(* IEC 61131-3 sources: volt/packages/volt-lsp-iec/test-corpus/pro2193/Device/Plc Logic/Application/09 Misc/Library Manager/L_MC1P_MotionControlBasic (part 7) *)

(* ---- L_MC1P_RESETMASTER_ETC.pou ---- *)
FUNCTION_BLOCK L_MC1P_RESETMASTER_ETC
VAR_INPUT
	XEXECUTE : BOOL;
	PSLAVE : POINTER TO ETCSlave;
END_VAR
VAR_OUTPUT
	XDONE : BOOL;
	XERROR : BOOL;
	XBUSY : BOOL;
	DWERROR : DWORD;
END_VAR
VAR
	XEXECUTEOLD : BOOL;
	WACTMASTERSTATE : INT;
	SETMASTERSTATE : L_ETC.L_ETC_SetMasterState;
	PMASTER : POINTER TO L_ETC.L_IODrvEtherCAT;
END_VAR
END_FUNCTION_BLOCK

METHOD ACYCLICACTION
END_METHOD

(* ---- L_MC1P_SAFETYCONTROLDECODER.pou ---- *)
FUNCTION_BLOCK L_MC1P_SAFETYCONTROLDECODER
VAR_INPUT
	XENABLE : BOOL;
	DWCONTROL : DWORD;
END_VAR
VAR_OUTPUT
	XBUSY : BOOL;
	XERROR : BOOL;
	EERRORID : L_IE1P_Error;
	XSTO_ACTIVE : BOOL;
	XSS1_ACTIVE : BOOL;
	XSS2_ACTIVE : BOOL;
	XSOS_ACTIVE : BOOL;
	XSLS1_ACTIVE : BOOL;
	XSLS2_ACTIVE : BOOL;
	XSLS3_ACTIVE : BOOL;
	XSLS4_ACTIVE : BOOL;
	XSDIPOS_ACTIVE : BOOL;
	XSDINEG_ACTIVE : BOOL;
	XSLI_ACTIVE : BOOL;
	XSSE_ACTIVE : BOOL;
	XES_ACTIVE : BOOL;
	XOMS_ACTIVE : BOOL;
	XRMS_ACTIVE : BOOL;
	XSBC_ACTIVE : BOOL;
	XMUT_ACTIVE : BOOL;
END_VAR
END_FUNCTION_BLOCK

(* ---- L_MC1P_SAFETYCONTROLENCODER.pou ---- *)
FUNCTION_BLOCK L_MC1P_SAFETYCONTROLENCODER
VAR_INPUT
	XENABLE : BOOL;
	XSTO_ACTIVE : BOOL;
	XSS1_ACTIVE : BOOL;
	XSS2_ACTIVE : BOOL;
	XSOS_ACTIVE : BOOL;
	XSLS1_ACTIVE : BOOL;
	XSLS2_ACTIVE : BOOL;
	XSLS3_ACTIVE : BOOL;
	XSLS4_ACTIVE : BOOL;
	XSDIPOS_ACTIVE : BOOL;
	XSDINEG_ACTIVE : BOOL;
	XSLI_ACTIVE : BOOL;
	XSSE_ACTIVE : BOOL;
	XES_ACTIVE : BOOL;
	XOMS_ACTIVE : BOOL;
	XRMS_ACTIVE : BOOL;
	XSBC_ACTIVE : BOOL;
	XMUT_ACTIVE : BOOL;
END_VAR
VAR_OUTPUT
	XBUSY : BOOL;
	XERROR : BOOL;
	EERRORID : L_IE1P_Error;
	DWCONTROL : DWORD;
END_VAR
END_FUNCTION_BLOCK

(* ---- L_MC1P_SAFETYIOSTATEDECODER.pou ---- *)
FUNCTION_BLOCK L_MC1P_SAFETYIOSTATEDECODER
VAR_INPUT
	XENABLE : BOOL;
	DWIOSTATE : DWORD;
END_VAR
VAR_OUTPUT
	XBUSY : BOOL;
	XERROR : BOOL;
	EERRORID : L_IE1P_Error;
	XSDIN1 : BOOL;
	XSDIN2 : BOOL;
	XSDIN3 : BOOL;
	XSDIN4 : BOOL;
	XAIS_DIGIN : BOOL;
	XAIE_DIGIN : BOOL;
	XIRS_DIGIN : BOOL;
	XIRL_DIGIN : BOOL;
	XAIS_SBUS : BOOL;
	XAIE_SBUS : BOOL;
	XSHOMSTART_SBUS : BOOL;
	XSHOMLOAD_SBUS : BOOL;
	XSDOUT1 : BOOL;
	XSDIN1A : BOOL;
	XSDIN1B : BOOL;
	XSDIN2A : BOOL;
	XSDIN2B : BOOL;
	XSDIN3A : BOOL;
	XSDIN3B : BOOL;
	XSDIN4A : BOOL;
	XSDIN4B : BOOL;
	XSDOUT1A : BOOL;
	XSDOUT1B : BOOL;
END_VAR
END_FUNCTION_BLOCK

(* ---- L_MC1P_SAFETYREADSTATUSWORDS.pou ---- *)
FUNCTION_BLOCK L_MC1P_SAFETYREADSTATUSWORDS EXTENDS L_MC1P_Template
VAR_INPUT
	XENABLE : BOOL;
END_VAR
VAR_OUTPUT
	XVALID : BOOL;
	XBUSY : BOOL;
	XERROR : BOOL;
	EERRORID : L_IE1P_Error;
	DWCONTROL : DWORD;
	DWSTATE : DWORD;
	DWIOSTATE : DWORD;
END_VAR
VAR
	XENABLEOLD : BOOL;
END_VAR
END_FUNCTION_BLOCK

(* ---- L_MC1P_SAFETYSTATEDECODER.pou ---- *)
FUNCTION_BLOCK L_MC1P_SAFETYSTATEDECODER
VAR_INPUT
	XENABLE : BOOL;
	DWSTATE : DWORD;
END_VAR
VAR_OUTPUT
	XBUSY : BOOL;
	XERROR : BOOL;
	EERRORID : L_IE1P_Error;
	XSLS1_OBSERVED : BOOL;
	XSLS2_OBSERVED : BOOL;
	XSLS3_OBSERVED : BOOL;
	XSLS4_OBSERVED : BOOL;
	XSMS_OBSERVED : BOOL;
	XSSM_WITHINLIMITS : BOOL;
	XSDIPOS_OBSERVED : BOOL;
	XSDINEG_OBSERVED : BOOL;
	XSLP1_OBSERVED : BOOL;
	XSLP2_OBSERVED : BOOL;
	XSLP3_OBSERVED : BOOL;
	XSLP4_OBSERVED : BOOL;
	XSCA1_WITHINLIMITS : BOOL;
	XSCA2_WITHINLIMITS : BOOL;
	XSCA3_WITHINLIMITS : BOOL;
	XSCA4_WITHINLIMITS : BOOL;
	XPDSSPOS_OBSERVED : BOOL;
	XPDSSNEG_OBSERVED : BOOL;
	XSOS_OBSERVED : BOOL;
	XSBC_ACTIVATED : BOOL;
	XSHOM_ACTIVE : BOOL;
	XSHOM_AVAILABLE : BOOL;
	XSAFESPEED_OK : BOOL;
	XSPEEDEQ0 : BOOL;
	XPOSDIRECTION : BOOL;
	XSLIPGT25 : BOOL;
	XSLIPGT50 : BOOL;
	XSLIPGT75 : BOOL;
	XERRORACTIVE : BOOL;
END_VAR
END_FUNCTION_BLOCK

(* ---- L_MC1P_SETAXISREFMASTERVALUES.pou ---- *)
FUNCTION_BLOCK L_MC1P_SETAXISREFMASTERVALUES
VAR_INPUT
	LRSETPOSIN : LREAL;
	LRSETVELIN : LREAL;
	LRSETACCIN : LREAL;
	LRTORQUEIN : LREAL;
	LRCYCLELENGTH : LREAL;
	ETRAVERSINGRANGE : L_MC1P_TraversingRange;
	XINTERPOLATEINPUTS : BOOL;
	LRINPUTCYCLETIME : LREAL := 0.001;
	EINTERPOLATIONMODE : L_MC1P_InterpolationMode := L_MC1P_InterpolationMode.linear;
	WDIRECTION : WORD;
	XACTIVATETELEGRAMLOSSDETECTION : BOOL;
	XSYNCPROCESSDATAEXPECTED : BOOL;
	XSYNCPROCESSDATAVALID : BOOL;
END_VAR
VAR_OUTPUT
	MASTERVALUES : L_MC1P_IAXIS_REF_MASTERVALUES;
	LRSETPOSOUT : LREAL;
	LRSETVELOUT : LREAL;
	LRSETACCOUT : LREAL;
	LRTORQUEOUT : LREAL;
END_VAR
VAR
	XINITDONE : BOOL := FALSE;
	LRSETPOSINOLD : LREAL;
	LRSETVELINOLD : LREAL;
	LRSETACCINOLD : LREAL;
	LRTORQUEINOLD : LREAL;
	LRSETPOSSTART : LREAL;
	LRSETVELSTART : LREAL;
	LRSETACCSTART : LREAL;
	LRTORQUESTART : LREAL;
	LRSETPOSEND : LREAL;
	LRSETVELEND : LREAL;
	LRSETACCEND : LREAL;
	LRTORQUEEND : LREAL;
	LRTASKCYCLE : LREAL := 0.001;
	LRINVTASKCYCLE : LREAL := 1000;
	LRACTCYCLE : LREAL;
	LRMAXCYCLE : LREAL;
	LRINVMAXCYCLE : LREAL;
	XSTARTINTERPOLATION : BOOL;
	LRPOSDIFF : LREAL;
	LRPOSDIFFOLD : LREAL;
	LRSETPOSSTARTOLD : LREAL;
	LRACC : LREAL;
	LRVEL : LREAL;
	FB_GETDIRECTION : L_MC1P_GetDirection;
	WEXTRAPOLATIONCOUNTER : WORD;
	WINTERPOLATIONCOUNTER : WORD;
	POSV : LREAL;
	C_COUNTERLIMIT : WORD := 1000;
	ACTACCELERATION : LREAL;
	ACTPOSITION : LREAL;
	ACTTORQUE : LREAL;
	ACTVELOCITY : LREAL;
	CYCLELENGTH : LREAL;
	FEEDCONSTANT : LREAL;
	GETMASTERID : POINTER TO BYTE;
	SETACCELERATIONFORSYNC : LREAL;
	SETPOSITIONFORSYNC : LREAL;
	SETTORQUEFORSYNC : LREAL;
	SETVELOCITYFORSYNC : LREAL;
	TASKCYCLE : LREAL;
	TRAVERSINGRANGE : L_MC1P_TraversingRange;
END_VAR
END_FUNCTION_BLOCK

METHOD GETDIRECTION : WORD
VAR_INPUT
	VALUESOURCE : MC_SOURCE;
END_VAR
END_METHOD

METHOD GETMASTERERROR : BOOL
VAR_OUTPUT
	EERRORID : L_IE1P_Error;
END_VAR
END_METHOD

METHOD GETSTEADYSTATE : POINTER TO L_MC1P_SteadyState
END_METHOD

METHOD FB_INIT : BOOL
VAR_INPUT
	BINITRETAINS : BOOL;
	BINCOPYCODE : BOOL;
END_VAR
END_METHOD

(* ---- L_MC1P_SETBASICPARAMETER.pou ---- *)
FUNCTION_BLOCK L_MC1P_SETBASICPARAMETER EXTENDS L_MC1P_Template
VAR_INPUT
	XENABLE : BOOL;
	XSETJOGPARAMETER : BOOL;
	LRJOGVEL : LREAL := 360;
	LRJOGACC : LREAL := 360;
	LRJOGDEC : LREAL := 1440;
	LRJOGJERK : LREAL := 0;
	XSETHALTPARAMETER : BOOL;
	LRHALTDEC : LREAL := 1800;
	LRHALTJERK : LREAL := 0;
	XSETQSPAPPLPARAMETER : BOOL;
	LRQSPAPPLDEC : LREAL := 3600.0;
	LRQSPAPPLJERK : LREAL := 0;
	XSETHOMEPOSITION : BOOL;
	LRHOMEPOSITION : LREAL;
	XSETHOMEPARAMETER : BOOL;
	SCHOMEPARAMETER : L_MC1P_HomeParameter := STRUCT(eHomeMode := L_MC1P_HomeMode.SetPositionDirect, eHomeStopMode := L_MC1P_HomeStopMode.StopPositioning, lrTargetPosition := 0, lrVelocity1 := 360.0, lrVelocity2 := 0, lrAcceleration1 := 720.0, lrAcceleration2 := 360.0, lrJerk := 7200.0, rTorqueLimit := 0.1, rTorqueTime := 1.0, dwTPConfig := 1, eStopModeDirection := MC_DIRECTION.mcCurrentDirection);
END_VAR
VAR_OUTPUT
	XBUSY : BOOL;
	XERROR : BOOL;
	EERRORID : L_IE1P_Error;
END_VAR
VAR
	ICACHEARRAYINITIDX : INT := -1;
	ICACHEARRAYFIRSTIDX : INT := 0;
	ICACHEARRAYLASTIDX : INT := 15;
	ADIRBPARAMETERS : ARRAY [iCacheArrayFirstIdx..iCacheArrayLastIdx] OF DINT;
	ALRRBVALUES : ARRAY [iCacheArrayFirstIdx..iCacheArrayLastIdx] OF LREAL;
	IRBACTIDX : INT := -1;
END_VAR
END_FUNCTION_BLOCK

METHOD SETBASICPARAMETER : DWORD
END_METHOD

METHOD WRITEPARAM : BOOL
VAR_INPUT
	PARAMETER : DINT;
	LRVALUE : LREAL;
	EWRITEERRORID : L_IE1P_Error;
END_VAR
END_METHOD

(* ---- L_MC1P_SETCONTROLMODE.pou ---- *)
FUNCTION_BLOCK L_MC1P_SETCONTROLMODE EXTENDS L_MC1P_Template
VAR_INPUT
	XEXECUTE : BOOL;
	ECONTROLMODE : L_MC1P_ControlModeSet := L_MC1P_ControlModeSet.PosCtrlDrive;
	XKEEPACTPOSPRIORFDB : BOOL := FALSE;
	XRESTARTPOSITIONING : BOOL := FALSE;
END_VAR
VAR_OUTPUT
	XDONE : BOOL;
	XBUSY : BOOL;
	XERROR : BOOL;
	EERRORID : L_IE1P_Error;
END_VAR
VAR
	FBSETCONTROLMODEINTERN : L_MC1P_SetControlMode_Internal;
END_VAR
END_FUNCTION_BLOCK

(* ---- L_MC1P_SETCONTROLMODE_INTERNAL.pou ---- *)
FUNCTION_BLOCK L_MC1P_SETCONTROLMODE_INTERNAL EXTENDS L_MC1P_Template_IntFB
VAR_INPUT
	XEXECUTE : BOOL;
	ECONTROLMODE : L_MC1P_ControlModeSet := L_MC1P_ControlModeSet.PosCtrlDrive;
	XKEEPACTPOSPRIORFDB : BOOL := FALSE;
	XRESTARTPOSITIONING : BOOL := FALSE;
END_VAR
VAR_OUTPUT
	XDONE : BOOL;
	XBUSY : BOOL;
	XERROR : BOOL;
	EERRORID : L_IE1P_Error;
END_VAR
VAR
	XEXECUTEOLD : BOOL;
	XRESETOUTPUT : BOOL;
END_VAR
END_FUNCTION_BLOCK

METHOD MAIN
VAR_IN_OUT
	AXIS : AXIS_REF;
	FBBASE : L_MC1P_Template_ForAxis;
END_VAR
END_METHOD

(* ---- L_MC1P_SETDCBRAKE.pou ---- *)
FUNCTION_BLOCK L_MC1P_SETDCBRAKE EXTENDS L_MC1P_Template
VAR_INPUT
	XENABLE : BOOL;
END_VAR
VAR_OUTPUT
	XBUSY : BOOL;
	XACTIVE : BOOL;
	XERROR : BOOL;
	EERRORID : L_IE1P_Error;
END_VAR
VAR
	XENABLEOLD : BOOL;
END_VAR
END_FUNCTION_BLOCK

(* ---- L_MC1P_SETEXTERNALENCODER.pou ---- *)
FUNCTION_BLOCK L_MC1P_SETEXTERNALENCODER EXTENDS L_MC1P_Template
VAR_INPUT
	ENCODER : L_MC1P_IEncoderInterface;
	XEXECUTE : BOOL;
END_VAR
VAR_OUTPUT
	XDONE : BOOL;
	XBUSY : BOOL;
	XERROR : BOOL;
	EERRORID : L_IE1P_Error;
END_VAR
VAR
	XEXECUTEOLD : BOOL;
	PAXISREALDRIVE : POINTER TO _AXIS_REF_REAL;
	PAXISREAL : POINTER TO _AXIS_REF_REAL;
	PXDUMMY : POINTER TO BOOL;
	PSDUMMY : POINTER TO STRING;
END_VAR
END_FUNCTION_BLOCK

(* ---- L_MC1P_SETFASTSTOP.pou ---- *)
FUNCTION_BLOCK L_MC1P_SETFASTSTOP EXTENDS L_MC1P_Template
VAR_INPUT
	XENABLE : BOOL;
END_VAR
VAR_OUTPUT
	XBUSY : BOOL;
	XACTIVE : BOOL;
	XERROR : BOOL;
	EERRORID : L_IE1P_Error;
END_VAR
VAR
	XENABLEOLD : BOOL;
	FBSETFASTSTOP : L_MC1P_SetFastStop_Internal;
END_VAR
END_FUNCTION_BLOCK

(* ---- L_MC1P_SETFASTSTOP_INTERNAL.pou ---- *)
FUNCTION_BLOCK L_MC1P_SETFASTSTOP_INTERNAL EXTENDS L_MC1P_Template_IntFB
VAR_INPUT
	XENABLE : BOOL;
END_VAR
VAR_OUTPUT
	XBUSY : BOOL;
	XACTIVE : BOOL;
	XERROR : BOOL;
	EERRORID : L_IE1P_Error;
END_VAR
VAR
	XENABLEOLD : BOOL;
END_VAR
END_FUNCTION_BLOCK

METHOD MAIN
VAR_IN_OUT
	AXIS : AXIS_REF;
	FBBASE : L_MC1P_Template_ForAxis;
END_VAR
END_METHOD

(* ---- L_MC1P_SETINERTIAADAPTVALUE.pou ---- *)
FUNCTION_BLOCK L_MC1P_SETINERTIAADAPTVALUE EXTENDS L_MC1P_Template
VAR_INPUT
	XENABLE : BOOL;
	LRINERTIAADAPTVALUE : LREAL := 1.0;
END_VAR
VAR_OUTPUT
	XBUSY : BOOL;
	XERROR : BOOL;
	EERRORID : L_IE1P_Error;
END_VAR
VAR
	PAXIS : POINTER TO _AXIS_REF_REAL;
	XENABLEOLD : BOOL;
END_VAR
END_FUNCTION_BLOCK

(* ---- L_MC1P_SETOVERRIDE_INTERNAL.pou ---- *)
FUNCTION_BLOCK L_MC1P_SETOVERRIDE_INTERNAL EXTENDS L_MC1P_Template_IntFB
VAR_INPUT
	ENABLE : BOOL;
	VELFACTOR : LREAL := 1.0;
	ACCFACTOR : LREAL := 1.0;
	JERKFACTOR : LREAL := 1.0;
END_VAR
VAR_OUTPUT
	ENABLED : BOOL;
	BUSY : BOOL;
	ERROR : BOOL;
	ERRORID : L_IE1P_Error;
END_VAR
VAR
	XENABLEOLD : BOOL;
	WDATAOLD : WORD;
END_VAR
END_FUNCTION_BLOCK

METHOD MAIN
VAR_IN_OUT
	AXIS : AXIS_REF;
	FBBASE : L_MC1P_Template_ForAxis;
END_VAR
END_METHOD

(* ---- L_MC1P_SETPOSCTRLADAPTVALUE.pou ---- *)
FUNCTION_BLOCK L_MC1P_SETPOSCTRLADAPTVALUE EXTENDS L_MC1P_Template
VAR_INPUT
	XENABLE : BOOL;
	LRPOSCTRLADAPTVALUE : LREAL := 1.0;
	EMODE : L_MC1P_PosCtrlAdaptMode := L_MC1P_PosCtrlAdaptMode.MotorAndLoad;
END_VAR
VAR_OUTPUT
	XBUSY : BOOL;
	XERROR : BOOL;
	EERRORID : L_IE1P_Error;
END_VAR
VAR
	ISTATE : INT := 0;
	DNPOSCTRLADAPTVAL : DINT;
	DNPOSCTRLADAPTVALOLD : DINT := 100;
	BYSDORETRYCOUNTER : BYTE;
	XWAITFORPARAMETERWRITEDONE : BOOL;
	WRITEPARAMETER : L_DCO_WriteDriveParameter;
	XCHECKCONFIG : BOOL;
	XUSEPDOINTERFACE : BOOL;
	WINDEX : WORD;
	BYSUBINDEX : BYTE;
	BYNROFBYTE : BYTE;
	XINITDONE : BOOL := FALSE;
	XWRITEINITPARAMETER : BOOL := TRUE;
	DNPARAMETERWRITEVALUE : DINT;
	PAXIS : POINTER TO _AXIS_REF_REAL;
	L_MC1P_CYCLICPARAMETERACCESSWRITE1 : L_MC1P_CyclicParameterAccessWrite;
	XENABLEFORDRIVE : BOOL;
	SDO_WRITE_TIME_OUT : UDINT := 10000;
	MAX_SDO_RETRIES : BYTE := 3;
END_VAR
END_FUNCTION_BLOCK

(* ---- L_MC1P_SETQUICKSTOP.pou ---- *)
FUNCTION_BLOCK L_MC1P_SETQUICKSTOP EXTENDS L_MC1P_Template
VAR_INPUT
	XENABLE : BOOL;
END_VAR
VAR_OUTPUT
	XBUSY : BOOL;
	XACTIVE : BOOL;
	XERROR : BOOL;
	EERRORID : L_IE1P_Error;
END_VAR
VAR
	XENABLEOLD : BOOL;
END_VAR
END_FUNCTION_BLOCK

(* ---- L_MC1P_SETQUICKSTOPAPPL.pou ---- *)
FUNCTION_BLOCK L_MC1P_SETQUICKSTOPAPPL EXTENDS L_MC1P_Template
VAR_INPUT
	XENABLE : BOOL;
END_VAR
VAR_OUTPUT
	XBUSY : BOOL;
	XACTIVE : BOOL;
	XERROR : BOOL;
	EERRORID : L_IE1P_Error;
END_VAR
VAR
	XENABLEOLD : BOOL;
	FBSETFASTSTOP : L_MC1P_SetFastStop_Internal;
END_VAR
END_FUNCTION_BLOCK

(* ---- L_MC1P_SETQUICKSTOPOPTION.pou ---- *)
FUNCTION_BLOCK L_MC1P_SETQUICKSTOPOPTION EXTENDS L_MC1P_Template
VAR_INPUT
	XEXECUTE : BOOL;
	EQUICKSTOPOPTION : L_MC1P_QuickStopOption := L_MC1P_QuickStopOption.StayInQSP;
END_VAR
VAR_OUTPUT
	XDONE : BOOL;
	XBUSY : BOOL;
	XERROR : BOOL;
	EERRORID : L_IE1P_Error;
END_VAR
VAR
	XEXECUTEOLD : BOOL;
	XRESETOUTPUT : BOOL;
	ISTATE : INT;
	WRITEPARAMETER : L_DCO_WriteDriveParameter;
	PAXISREAL : POINTER TO _AXIS_REF_REAL;
	PWDUMMY : POINTER TO WORD;
END_VAR
END_FUNCTION_BLOCK

(* ---- L_MC1P_SETSETVALUEMANIPULATOR.pou ---- *)
FUNCTION_BLOCK L_MC1P_SETSETVALUEMANIPULATOR EXTENDS L_MC1P_ManipulationBase
VAR_INPUT
	XIGNOREFILTERONSTOP : BOOL;
END_VAR
VAR
	XUSEFILTERASMASTERVALUE_INT : BOOL := TRUE;
	XUSEFILTERASMASTERSOURCE : BOOL := TRUE;
	IGNOREFILTERONSTOP : BOOL;
	USEFILTERVALUESFORSYNC : BOOL;
END_VAR
END_FUNCTION_BLOCK

METHOD CALLCYCLIC2
VAR_IN_OUT
	AXIS : Axis_REf;
END_VAR
END_METHOD

METHOD CONNECTTOAXIS
VAR_IN_OUT
	AXIS : Axis_Ref;
END_VAR
END_METHOD

METHOD DISCONNECTFROMAXIS
VAR_IN_OUT
	AXIS : Axis_Ref;
END_VAR
END_METHOD

METHOD READINPUTS2
VAR_IN_OUT
	AXIS : Axis_REf;
END_VAR
END_METHOD

METHOD RESETOUTPUTS2
VAR_IN_OUT
	AXIS : Axis_REf;
END_VAR
END_METHOD

METHOD CALCULATE2
VAR_IN_OUT
	AXIS : Axis_REf;
END_VAR
END_METHOD

METHOD CHECKINPUTDATA2
VAR_IN_OUT
	AXIS : Axis_REf;
END_VAR
END_METHOD

METHOD ENABLEEXIT2
VAR_IN_OUT
	AXIS : Axis_REf;
END_VAR
END_METHOD

METHOD ENABLEINIT2
VAR_IN_OUT
	AXIS : Axis_REf;
END_VAR
END_METHOD

METHOD FILTERSTARTCONDITION
VAR_INPUT
	LRSETPOS : LREAL;
	LRSETVEL : LREAL;
	LRSETACC : LREAL;
END_VAR
VAR_IN_OUT
	AXIS : Axis_ref;
END_VAR
END_METHOD

METHOD LOADOFFSET2
VAR_INPUT
	OFFSET : LREAL;
END_VAR
VAR_IN_OUT
	AXIS : Axis_REf;
END_VAR
END_METHOD

METHOD RESET2
VAR_IN_OUT
	AXIS : Axis_REf;
END_VAR
END_METHOD

METHOD CALLCYCLIC
END_METHOD

METHOD READINPUTS
END_METHOD

METHOD RESETOUTPUTS
END_METHOD

METHOD CALCULATE
END_METHOD

METHOD CHECKINPUTDATA
END_METHOD

METHOD ENABLEEXIT
END_METHOD

METHOD ENABLEINIT
END_METHOD

METHOD LOADOFFSET
VAR_INPUT
	OFFSET : LREAL;
END_VAR
END_METHOD

METHOD RESET
END_METHOD

(* ---- L_MC1P_SETSPEEDCTRLADAPTVALUE.pou ---- *)
FUNCTION_BLOCK L_MC1P_SETSPEEDCTRLADAPTVALUE EXTENDS L_MC1P_Template
VAR_INPUT
	XENABLE : BOOL;
	LRSPEEDCTRLADAPTVALUE : LREAL := 1.0;
END_VAR
VAR_OUTPUT
	XBUSY : BOOL;
	XERROR : BOOL;
	EERRORID : L_IE1P_Error;
END_VAR
VAR
	ISTATE : INT := 0;
	DNSPEEDCTRLADAPTVAL : DINT;
	DNSPEEDCTRLADAPTVALOLD : DINT := 100;
	BYSDORETRYCOUNTER : BYTE;
	XWAITFORPARAMETERWRITEDONE : BOOL;
	WRITEPARAMETER : L_DCO_WriteDriveParameter;
	XCHECKCONFIG : BOOL;
	XUSEPDOINTERFACE : BOOL;
	WINDEX : WORD;
	BYSUBINDEX : BYTE;
	BYNROFBYTE : BYTE;
	XINITDONE : BOOL := FALSE;
	XWRITEINITPARAMETER : BOOL := TRUE;
	DNPARAMETERWRITEVALUE : DINT;
	PAXIS : POINTER TO _AXIS_REF_REAL;
	L_MC1P_CYCLICPARAMETERACCESSWRITE1 : L_MC1P_CyclicParameterAccessWrite;
	SDO_WRITE_TIME_OUT : UDINT := 10000;
	MAX_SDO_RETRIES : BYTE := 3;
END_VAR
END_FUNCTION_BLOCK

(* ---- L_MC1P_SETSPEEDCTRLLOADVALUE.pou ---- *)
FUNCTION_BLOCK L_MC1P_SETSPEEDCTRLLOADVALUE EXTENDS L_MC1P_Template
VAR_INPUT
	XENABLE : BOOL;
	LRSPEEDCTRLLOADVALUE : LREAL := 1.0;
END_VAR
VAR_OUTPUT
	XBUSY : BOOL;
	XERROR : BOOL;
	EERRORID : L_IE1P_Error;
END_VAR
VAR
	XENABLEOLD : BOOL;
	PAXIS : POINTER TO _AXIS_REF_REAL;
END_VAR
END_FUNCTION_BLOCK

(* ---- L_MC1P_SETTORQUELIMIT.pou ---- *)
FUNCTION_BLOCK L_MC1P_SETTORQUELIMIT EXTENDS L_MC1P_Template
VAR_INPUT
	XENABLE : BOOL;
	XSETTORQUELIMITPOS : BOOL;
	LRTORQUELIMITPOS : LREAL;
	XSETTORQUELIMITNEG : BOOL;
	LRTORQUELIMITNEG : LREAL;
	XTORQUEINPUTASPERCENT : BOOL;
END_VAR
VAR_OUTPUT
	XBUSY : BOOL;
	XERROR : BOOL;
	EERRORID : L_IE1P_Error;
END_VAR
VAR
	XENABLEOLD : BOOL;
	PAXIS : POINTER TO _AXIS_REF_REAL;
	PXDUMMY : POINTER TO BOOL;
	LRTMP : LREAL;
END_VAR
END_FUNCTION_BLOCK

METHOD CHECKTORQUEVALUE : LREAL
VAR_INPUT
	LRTORQUE : LREAL;
	LRDEFAULTTORQUE : LREAL;
END_VAR
VAR_IN_OUT
	AXIS : AXIS_REF;
END_VAR
END_METHOD

(* ---- L_MC1P_SETTORQUEOFFSET.pou ---- *)
FUNCTION_BLOCK L_MC1P_SETTORQUEOFFSET EXTENDS L_MC1P_Template
VAR_INPUT
	XENABLE : BOOL;
	LRTORQUE : LREAL;
	EPRECONTROLMODE : L_MC1P_PreControlMode := L_MC1P_PreControlMode.AdditiveOffsetTorque;
END_VAR
VAR_OUTPUT
	XBUSY : BOOL;
	XERROR : BOOL;
	EERRORID : L_IE1P_Error;
END_VAR
VAR
	XENABLEOLD : BOOL;
END_VAR
END_FUNCTION_BLOCK

(* ---- L_MC1P_SIMMECHANIC.pou ---- *)
FUNCTION_BLOCK L_MC1P_SIMMECHANIC EXTENDS L_MC1P_SimMechanicBase
VAR_INPUT
	SCPAR : L_MC1P_ParMechanic;
END_VAR
VAR
	XLIMITEDPOS : BOOL;
	LRFRICTORQUE : LREAL;
	LRACTVEL_INT : LREAL;
	LRACTACC_INT : LREAL;
	LRACTPOS_INT : LREAL;
	LRINERTIAINV : LREAL;
	LOADFDB : LREAL;
END_VAR
END_FUNCTION_BLOCK

METHOD CALLMECHANICSIMULATION : BOOL
VAR_INPUT
	XBRAKERELEASED : BOOL;
	LRACTTORQUE : LREAL;
	LRTASKCYCLESYSSIM : LREAL;
	LRINVTASKCYCLESYSSIM : LREAL;
END_VAR
VAR_OUTPUT
	LRACTPOS : LREAL;
	LRACTVEL : LREAL;
END_VAR
END_METHOD

METHOD SCALEPARAMETER
END_METHOD

METHOD SETSTARTPOSITION : BOOL
VAR_INPUT
	LRPOS : LREAL;
END_VAR
END_METHOD

(* ---- L_MC1P_SIMMECHANIC2MS.pou ---- *)
FUNCTION_BLOCK L_MC1P_SIMMECHANIC2MS EXTENDS L_MC1P_SimMechanicBase
VAR_INPUT
	SCPAR : L_MC1P_ParMechanic2ms;
END_VAR
VAR
	LRFRICTORQUEMOT : LREAL;
	LRFRICTORQUELOAD : LREAL;
	XZEROCROSSINGBRAKECLOSED : BOOL := FALSE;
	ALRX_DIFF : ARRAY [0..3] OF LREAL;
	ALRX : ARRAY [0..3] OF LREAL;
	ALRA : ARRAY [0..1, 0..3] OF LREAL;
	LRINERTIAINV : LREAL;
	LRINERTIA2INV : LREAL;
	LREIGENFREQUENCYSQR : LREAL;
	LRPHITORSION : LREAL;
	LROMEGATORSION : LREAL;
	LRALPHATORSION : LREAL;
	LRVISCOSEFACTORMOT : LREAL;
	LRCOULOMBFACTORMOT : LREAL;
	LRVISCOSEFACTORLOAD : LREAL;
	LRCOULOMBFACTORLOAD : LREAL;
	XUSESIMPLIFIEDMODEL : BOOL;
	LOADFDB : LREAL;
END_VAR
END_FUNCTION_BLOCK

METHOD CALLMECHANICSIMULATION : BOOL
VAR_INPUT
	XBRAKERELEASED : BOOL;
	LRACTTORQUE : LREAL;
	LRTASKCYCLESYSSIM : LREAL;
	LRINVTASKCYCLESYSSIM : LREAL;
END_VAR
VAR_OUTPUT
	LRACTPOS : LREAL;
	LRACTVEL : LREAL;
END_VAR
END_METHOD

METHOD SCALEPARAMETER
END_METHOD

METHOD SETSTARTPOSITION : BOOL
VAR_INPUT
	LRPOS : LREAL;
END_VAR
END_METHOD

(* ---- L_MC1P_SIMMECHANIC2MS_BACKLASH.pou ---- *)
FUNCTION_BLOCK L_MC1P_SIMMECHANIC2MS_BACKLASH EXTENDS L_MC1P_SimMechanicBase
VAR_INPUT
	SCPAR : L_MC1P_ParMechanic2ms_Backlash;
END_VAR
VAR
	LRFRICTORQUEMOT : LREAL;
	LRFRICTORQUELOAD : LREAL;
	XZEROCROSSINGBRAKECLOSED : BOOL := FALSE;
	ALRX_DIFF : ARRAY [0..2] OF LREAL;
	ALRX : ARRAY [0..4] OF LREAL;
	ALRA : REFERENCE TO ARRAY [0..2, 0..4] OF LREAL;
	ALRA_CONTACT : ARRAY [0..2, 0..4] OF LREAL;
	ALRA_ZERO : ARRAY [0..2, 0..4] OF LREAL;
	ECONTACT : L_MC1P_BacklashContactState;
	LRTHETA : LREAL;
	LRDTHETA : LREAL;
	LRD_DIV_C : LREAL;
	LRINERTIAINV : LREAL;
	LRINERTIA2INV : LREAL;
	LRVISCOSEFACTORMOT : LREAL;
	LRCOULOMBFACTORMOT : LREAL;
	LRVISCOSEFACTORLOAD : LREAL;
	LRCOULOMBFACTORLOAD : LREAL;
	LREIGENFREQUENCYSQR : LREAL;
	XUSESIMPLIFIEDMODEL : BOOL;
	FBSIMPLIFIEDHYSTERESIS : L_UMTP_Hysteresis;
	LOADFDB : LREAL;
END_VAR
END_FUNCTION_BLOCK

METHOD CALLMECHANICSIMULATION : BOOL
VAR_INPUT
	XBRAKERELEASED : BOOL;
	LRACTTORQUE : LREAL;
	LRTASKCYCLESYSSIM : LREAL;
	LRINVTASKCYCLESYSSIM : LREAL;
END_VAR
VAR_OUTPUT
	LRACTPOS : LREAL;
	LRACTVEL : LREAL;
END_VAR
END_METHOD

METHOD SCALEPARAMETER
END_METHOD

METHOD SETSTARTPOSITION : BOOL
VAR_INPUT
	LRPOS : LREAL;
END_VAR
END_METHOD

(* ---- L_MC1P_SIMMECHANIC3MS.pou ---- *)
FUNCTION_BLOCK L_MC1P_SIMMECHANIC3MS EXTENDS L_MC1P_SimMechanicBase
VAR_INPUT
	SCPAR : L_MC1P_ParMechanic3ms;
END_VAR
VAR
	LRFRICTORQUE : LREAL;
	ALRX_DIFF : ARRAY [0..5] OF LREAL;
	ALRX : ARRAY [0..5] OF LREAL;
	ALRA : ARRAY [0..3, 0..5] OF LREAL;
	LRINERTIAINV : LREAL;
	LRINERTIA2INV : LREAL;
	LRINERTIA3INV : LREAL;
	LOADFDB : LREAL;
END_VAR
END_FUNCTION_BLOCK

METHOD CALLMECHANICSIMULATION : BOOL
VAR_INPUT
	XBRAKERELEASED : BOOL;
	LRACTTORQUE : LREAL;
	LRTASKCYCLESYSSIM : LREAL;
	LRINVTASKCYCLESYSSIM : LREAL;
END_VAR
VAR_OUTPUT
	LRACTPOS : LREAL;
	LRACTVEL : LREAL;
END_VAR
END_METHOD

METHOD SCALEPARAMETER
END_METHOD

METHOD SETSTARTPOSITION : BOOL
VAR_INPUT
	LRPOS : LREAL;
END_VAR
END_METHOD

(* ---- L_MC1P_SIMMECHANICBASE.pou ---- *)
FUNCTION_BLOCK L_MC1P_SIMMECHANICBASE
VAR
	XPARAMETERVALID : BOOL;
END_VAR
END_FUNCTION_BLOCK

METHOD CALCFRICTIONTORQUE : LREAL
VAR_INPUT
	LRVISCOSEFACTOR : LREAL;
	LRCOULOMBFACTOR : LREAL;
	LRCOULOMBSLOPE : LREAL;
	LRVEL : LREAL;
END_VAR
END_METHOD

(* ---- L_MC1P_SIMMOTORCTRL.pou ---- *)
FUNCTION_BLOCK L_MC1P_SIMMOTORCTRL
VAR_INPUT
	ITFMECHANICSIMULATION : L_MC1P_IMechanicSimulation;
	LRBUSCYCLE : LREAL;
END_VAR
VAR_IN_OUT
	SCPAR : L_MC1P_AxisSimulationSdoData;
	SCINPUTDATA : L_MC1P_AxisSimulationPDOdataToDriveScaled;
	SCOUTPUTDATA : L_MC1P_AxisSimulationPDOdataFromDriveScaled;
	SCIODATA : L_MC1P_AxisSimIOData;
	SCPARGENERAL : L_MC1P_ParGeneralMechanic;
END_VAR
VAR
	XREGULATORON : BOOL;
	XREGULATORONOLD : BOOL;
	XQSPACTIVE : BOOL;
	XERRORACTIVE : BOOL;
	XERRORREACTIONACTIVE : BOOL;
	XSTOACTIVE : BOOL := FALSE;
	LRPOSCTRL_VP : LREAL := 20;
	LRDRZCTRL_VP : LREAL := 0.01;
	LRDRZCTRL_TN : LREAL := 0.012;
	LRFILTERTIMEACTVEL : LREAL := 0.001;
	LRPT1KOEFFVELFILTER : LREAL;
	LRPOSCTRLOUTPUTLIMITATION : LREAL;
	LRMAXMOTORSPEED : LREAL := (((6075 / 60) * 2) * Math.PI);
	LRADDSPEEDLIMITATION : LREAL := 0;
	LRMAXTORQUEMOTOR : LREAL := 10;
	LRPOSTORQUELIMIT : LREAL;
	LRNEGTORQUELIMIT : LREAL;
	LRIANTEIL_DRZCTRL : LREAL;
	LRIANTEIL_CST2 : LREAL;
	XSPEEDCTRLLIMITED : BOOL;
	XPOSCTRLLIMITED : BOOL;
	LRSETVEL_POSCTRL : LREAL;
	XTORQUELIMITED : BOOL;
	LRSETTORQUE : LREAL;
	XSPEEDSETPOINTLIMITED : BOOL;
	XSPEEDSETPOINT2LIMITED : BOOL;
	XUPPERSPEEDLIMITACTIVE : BOOL;
	XLOWERSPEEDLIMITACTIVE : BOOL;
	LRACTTORQUEMOTOR : LREAL;
	LRACTPOSMECHANIC : LREAL;
	LRACTVELMECHANIC : LREAL;
	XRELEASEBRAKEOUT : BOOL := FALSE;
	XBRAKERELEASED : BOOL;
	XBRAKERELEASED_CIASTATE : BOOL;
	LRACTBRAKETIME : LREAL;
	XBRAKELOGIKACTIVE : BOOL;
	XBRAKEFREEZESETVALUES : BOOL;
	LRSETPOSFREEZE : LREAL;
	WCIASTATEBRAKEMASK : WORD;
	LRBRAKEDELAYTIMER : LREAL;
	XBRAKEOPENINGACTIVE : BOOL;
	XBRAKECLOSINGACTIVE : BOOL;
	EBRAKELOGICSTATE : L_MC1P_BrakeLogicState;
	XLOADBRAKETORQUE : BOOL;
	LRBRAKELOADINGTORQUE : LREAL;
	UICIACTRL_INTERN : UINT;
	UICIASTATUSWORD_INTERN : UINT;
	LRSETPOS_INT : LREAL;
	LRSETVEL_INT : LREAL;
	LRSETTORQUE_INT : LREAL;
	LRSETTORQUE_DRZCTRL : LREAL;
	LRSETPOSOLD : LREAL;
	LRSETVELOLD : LREAL;
	LRSETTORQUEOLD : LREAL;
	LRACTFOLLOWINGERROR_INT : LREAL;
	LRPOSWINDOWREACHED : LREAL;
	ISYSTEMSIMCOUNTER : INT;
	ESYSTEMSIMKHZ : L_MC1P_SimAxisCycleTime := L_MC1P_SimAxisCycleTime.TaskCycle_64kHz;
	EPOSCTRLKHZ : L_MC1P_SimAxisCycleTime := L_MC1P_SimAxisCycleTime.TaskCycle_16kHz;
	EDRZCTRLKHZ : L_MC1P_SimAxisCycleTime := L_MC1P_SimAxisCycleTime.TaskCycle_16kHz;
	ECURRCTRLKHZ : L_MC1P_SimAxisCycleTime := L_MC1P_SimAxisCycleTime.TaskCycle_16kHz;
	LRINVTASKCYCLESYSSIM : LREAL;
	LRTASKCYCLESYSSIM : LREAL;
	LRINVTASKCYCLECURRCTRL : LREAL;
	LRTASKCYCLECURRCTRL : LREAL;
	LRINVSAMPLESPERPLCCYCLE : LREAL;
	LRINVTASKCYCLEDRZCTRL : LREAL;
	LRTASKCYCLEDRZCTRL : LREAL;
	LRTASKCYCLEDRZCTRLDIVTNN : LREAL;
	ISAMPLESPERPLCCYCLE : INT;
	ISAMPLERATIOCURRCTRL : INT;
	ISAMPLERATIODRZCTRL : INT;
	ISAMPLERATIOPOSCTRL : INT;
	LRSAMPLERATIOCURRCTRL : LREAL;
	LRSAMPLERATIODRZCTRL : LREAL;
	LRSAMPLERATIOPOSCTRL : LREAL;
	LRRESOLUTION_INT : LREAL;
	LRINVRESOLUTION_INT : LREAL;
	XINIT : BOOL := FALSE;
	LRQSPDECDELTA : LREAL;
	LRDELTAVELACC : LREAL;
	LRDELTAVELDEC : LREAL;
	LRSETVELRAMP : LREAL;
	RNDGEN : L_UMTP_RandomGenerator;
	LRMAXNOISE_POSITION : LREAL := 6E-05;
	LRMAXNOISE_TORQUE : LREAL := 0.001;
	XGAUSIAN : BOOL := TRUE;
	LRMEASUREDPOS : LREAL;
	LRMEASUREDVEL : LREAL;
	LRMEASUREDACC : LREAL;
	LRMEASUREDTORQUE : LREAL;
	LRMEASUREDPOSOLD : LREAL;
	LRMEASUREDVELOLD : LREAL;
	WQSPSTEP : WORD;
	QSPPOS : LREAL;
	SIMTOUCHPROBE : L_MC1P_SimTouchProbe;
	PT2_CURRENT : L_USPP_PT2Filter;
	LRCURRCTRLPT2TT_LRA : LREAL;
	LRCURRCTRLPT2TT_LRB : LREAL;
	MEMDEADTIME : L_UBUP_MemoryProvider20Lreal;
	FB_DEADTIME : L_USPP_DeadTimeInt;
	ALRCURRCTRLDELAYBUFFER : ARRAY [0..19] OF LREAL;
	WCURRCTRLDELAYBUFFERSIZE : WORD := 20;
	WCURRCTRLDELAY : WORD;
	WCURRCTRLDELAYIDX : WORD;
	LRCURRCTRLDELAYSUBCYCLE : LREAL;
	XCURRCTRLDELAYINITIALIZED : BOOL;
	PAWDUMMY : POINTER TO ARRAY [1..2] OF UINT;
	LRREVPERINK : LREAL;
	CWNOTREADYTOSWITCHON : WORD := 2#0;
	CWSWITCHONDISABLED : WORD := 2#1000000;
	CWREADYTOSWITCHON : WORD := 2#100001;
	CWSWITCHEDON : WORD := 2#100011;
	CWOPERATIONENABLED : WORD := 2#100111;
	CWQSPACTIVE : WORD := 2#111;
	CWFAULTREACTIONACTIVE : WORD := 2#1111;
	CWFAULT : WORD := 2#1000;
	CWSTATEMASK : WORD := 2#1101111;
END_VAR
END_FUNCTION_BLOCK

METHOD BRAKELOGIC : BOOL
VAR_INPUT
	XREGULATORON : BOOL;
	UIBRAKEMODE : UINT;
END_VAR
VAR_OUTPUT
	WCIASTATEOUT : WORD;
	WCIACTRLOUT : WORD;
END_VAR
VAR_IN_OUT
	SCPAR : L_MC1P_AxisSimulationSdoData;
	SCOUTPUTDATA : L_MC1P_AxisSimulationPDOdataFromDriveScaled;
	SCINPUTDATA : L_MC1P_AxisSimulationPDOdataToDriveScaled;
	XRELEASEBRAKEOUT : BOOL;
	XBRAKEOUTRELEASED : BOOL;
	WCIACTRLIN : WORD;
END_VAR
END_METHOD

METHOD CIASTATEMACHINE
VAR_OUTPUT
	XOPERATIONENABLED : BOOL;
	XFAULTACTIVE : BOOL;
END_VAR
VAR_IN_OUT
	WCIACTRLWORD : WORD;
	WCIASTATUSWORD : WORD;
END_VAR
END_METHOD

METHOD INIT : BOOL
END_METHOD

METHOD INITCYCLE : BOOL
END_METHOD

METHOD SETSTARTPOSITION : BOOL
VAR_INPUT
	LRPOS : LREAL;
END_VAR
END_METHOD

METHOD MEASUREACTVALUES
END_METHOD

METHOD CST_DRZ_KLAMMER
END_METHOD

METHOD CALC_REGULATOR
VAR_IN_OUT
	SCPAR : L_MC1P_AxisSimulationSdoData;
	SCINPUTDATA : L_MC1P_AxisSimulationPDOdataToDriveScaled;
END_VAR
END_METHOD

METHOD CALCULATETORQUE
END_METHOD

METHOD DRZCONTROLLER
END_METHOD

METHOD DRZREGLER : LREAL
VAR_INPUT
	LRSETDRZ : LREAL;
	LRPOSTORQUELIMIT : LREAL;
	LRNEGTORQUELIMIT : LREAL;
END_VAR
VAR_OUTPUT
	XSPEEDCTRLLIMITED : BOOL;
	XSPEEDSETPOINTLIMITED : BOOL;
END_VAR
VAR_IN_OUT
	LRIANTEIL_DRZCTRL : LREAL;
END_VAR
END_METHOD

METHOD INTERPOLATESETVALUES
VAR_IN_OUT
	SCINPUTDATA : L_MC1P_AxisSimulationPDOdataToDriveScaled;
END_VAR
END_METHOD

METHOD POSCONTROLLER
END_METHOD

METHOD BRAKEDYNAMICS
VAR_IN_OUT
	SCPARGENERAL : L_MC1P_ParGeneralMechanic;
END_VAR
END_METHOD

(* ---- L_MC1P_SIMTOUCHPROBE.pou ---- *)
FUNCTION_BLOCK L_MC1P_SIMTOUCHPROBE
VAR_INPUT
	UITPFUNCTION : UINT;
END_VAR
VAR_IN_OUT
	SCIODATA : L_MC1P_AxisSimIOData;
	SCOUTPUTDATA : L_MC1P_AxisSimulationPDOdataFromDriveScaled;
END_VAR
VAR
	XSETTP1OLD : BOOL;
	XSETTP2OLD : BOOL;
	XTPDETECTION1NOTDONE : BOOL := TRUE;
	XTPDETECTION2NOTDONE : BOOL := TRUE;
	ATPFUNCTION : ARRAY [1..2] OF BYTE;
	ATPSTATUS : ARRAY [1..2] OF BYTE;
	PWDUMMY : POINTER TO WORD;
	LRACTPOS : LREAL;
	LRACTPOSOLD : LREAL;
	LRTPPOS1 : LREAL;
	LRTPPOS2 : LREAL;
	LRTPNEG1 : LREAL;
	LRTPNEG2 : LREAL;
END_VAR
END_FUNCTION_BLOCK

METHOD HANDLETPLOGIC : BOOL
VAR_INPUT
	XTP : BOOL;
	BYTPFUNCTION : BYTE;
END_VAR
VAR_IN_OUT
	XTPSAVE : BOOL;
	XTPDETECTIONNOTDONE : BOOL;
	BYTPSTATUS : BYTE;
	LRTPPOS : LREAL;
	LRTPNEG : LREAL;
END_VAR
END_METHOD

(* ---- L_MC1P_STACKCONTROLARRAY.pou ---- *)
FUNCTION_BLOCK L_MC1P_STACKCONTROLARRAY
VAR_INPUT
	IMAXLEGTH : INT := 100;
	XSET : BOOL;
	XGET : BOOL;
END_VAR
VAR_OUTPUT
	XSTACKISFULL : BOOL;
	XSTACKISEMPTY : BOOL := TRUE;
	ISTACKLEGTH : INT := 0;
	ISTACKSTARTPOS : INT := 0;
	ISTACKENDPOS : INT := 0;
	IGETPOS : INT;
	ISETPOS : INT;
END_VAR
VAR
	XSET_OLD : BOOL;
	XGET_OLD : BOOL;
	ILATESTPOS : INT;
	IOLDESTPOS : INT;
END_VAR
END_FUNCTION_BLOCK

METHOD CALL_RESET
END_METHOD

METHOD GET_ELEMENT : INT
END_METHOD

METHOD GET_ELEMENTLATEST : INT
END_METHOD

METHOD SET_ELEMENT : INT
END_METHOD

METHOD SET_ELEMENTOLDEST : INT
END_METHOD

(* ---- L_MC1P_STEADYSTATE.pou ---- *)
FUNCTION_BLOCK L_MC1P_STEADYSTATE EXTENDS L_MC1P_Changeable
VAR
	EUNSTEADYREASON : L_MC1P_UnSteadyReason;
	LRSETPOSOFFSET : LREAL := 0;
	LRSETVELOFFSET : LREAL := 0;
	LRSETACCOFFSET : LREAL := 0;
	LRACTPOSOFFSET : LREAL := 0;
	LRACTVELOFFSET : LREAL := 0;
	LRACTACCOFFSET : LREAL := 0;
	LRSETPOSSTORED : LREAL := 0;
	LRSETVELSTORED : LREAL := 0;
	LRSETACCSTORED : LREAL := 0;
	LRACTPOSSTORED : LREAL := 0;
	LRACTVELSTORED : LREAL := 0;
	LRACTACCSTORED : LREAL := 0;
	ACTACCOFFSET : LREAL;
	ACTPOSOFFSET : LREAL;
	ACTVELOFFSET : LREAL;
	SETACCOFFSET : LREAL;
	SETPOSOFFSET : LREAL;
	SETVELOFFSET : LREAL;
	UNSTEADYREASON : L_MC1P_UnSteadyReason;
END_VAR
END_FUNCTION_BLOCK

METHOD STOREVALUES
VAR_INPUT
	LRSETPOS : LREAL := 0;
	LRSETVEL : LREAL := 0;
	LRSETACC : LREAL := 0;
	LRACTPOS : LREAL := 0;
	LRACTVEL : LREAL := 0;
	LRACTACC : LREAL := 0;
END_VAR
END_METHOD

METHOD UNSTEADYEVENT : BOOL
VAR_INPUT
	EUNSTEADYREASON : L_MC1P_UnSteadyReason;
	LRSETPOS : LREAL := 0;
	LRSETVEL : LREAL := 0;
	LRSETACC : LREAL := 0;
	LRACTPOS : LREAL := 0;
	LRACTVEL : LREAL := 0;
	LRACTACC : LREAL := 0;
END_VAR
END_METHOD

(* ---- L_MC1P_STOP_INTERNAL.pou ---- *)
FUNCTION_BLOCK L_MC1P_STOP_INTERNAL EXTENDS L_MC1P_Template_IntFB
VAR_INPUT
	EXECUTE : BOOL;
	DECELERATION : LREAL;
	JERK : LREAL;
END_VAR
VAR_OUTPUT
	DONE : BOOL;
	BUSY : BOOL;
	COMMANDABORTED : BOOL;
	ERROR : BOOL;
	ERRORID : L_IE1P_Error;
END_VAR
VAR
	XSTART : BOOL;
	EXECUTEOLD : BOOL;
	PG : REFERENCE TO L_MC1P_PosProfiler;
	SCPARAM : L_MC1P_ProfileParameter;
	WFUNID : WORD;
	XRESETOUTPUT : BOOL;
	EACTSTATE : L_MC1P_AXIS_STATE;
	XSUPERIMPOSED : BOOL;
	XDONEOLD : BOOL;
	XWARNING : BOOL;
	EWARNINGID : L_IE1P_Error;
	XWARNINGOLD : BOOL;
	EWARNINGIDOLD : L_IE1P_Error;
	LRDECINT : LREAL;
	LRJERKINT : LREAL;
	XUSED : BOOL;
	XPOSPROFILERINUSE : BOOL;
	POSPROFILERINUSE : BOOL;
	REMAININGTIMEOFPROFILE : LREAL;
	REMAININGTIMEOFPROFILEAVAILABLE : BOOL;
END_VAR
END_FUNCTION_BLOCK

METHOD MAIN
VAR_IN_OUT
	AXIS : AXIS_REF;
	FBBASE : L_MC1P_Template_ForAxis;
END_VAR
END_METHOD

METHOD RESET
VAR_IN_OUT
	FBBASE : L_MC1P_Template_ForAxis;
END_VAR
END_METHOD

(* ---- L_MC1P_SUSPENDFOLLOWINGERROR.pou ---- *)
FUNCTION_BLOCK L_MC1P_SUSPENDFOLLOWINGERROR EXTENDS L_MC1P_Template
VAR_INPUT
	XENABLE : BOOL;
END_VAR
VAR_OUTPUT
	XBUSY : BOOL;
	XERROR : BOOL;
	EERRORID : L_IE1P_Error;
END_VAR
VAR
	XENABLEOLD : BOOL := FALSE;
END_VAR
END_FUNCTION_BLOCK

(* ---- L_MC1P_TEMPLATE.pou ---- *)
FUNCTION_BLOCK L_MC1P_TEMPLATE EXTENDS L_MC1P_Template_ForAxis
VAR_IN_OUT
	AXIS : AXIS_REF;
END_VAR
VAR
	SINSTANCESTR : STRING;
	DISABLEERRORRESET : BOOL;
END_VAR
END_FUNCTION_BLOCK

METHOD FB_GETERRORITFID : DWORD
END_METHOD

METHOD FB_GETINSTSTRPOINTER : POINTER TO STRING
END_METHOD

METHOD FB_RESETERROR
VAR_INPUT
	XERROR : BOOL;
	WERRORID : WORD;
END_VAR
END_METHOD

METHOD FB_RESETINT
END_METHOD

METHOD FB_SETERROR
VAR_INPUT
	WERRORID : L_IE1P_Error := 0;
	XSETERRORSTOP : BOOL := FALSE;
END_VAR
END_METHOD

METHOD FB_SETERRORANDREACTION
VAR_INPUT
	WERRORID : L_IE1P_Error := 0;
	EERRORREACTION : L_IE1P_SeverityLevel := L_IE1P_SeverityLevel.NO_RESPONSE;
END_VAR
END_METHOD

METHOD FB_INIT : BOOL
VAR_INPUT
	BINITRETAINS : BOOL;
	BINCOPYCODE : BOOL;
END_VAR
END_METHOD

(* ---- L_MC1P_TEMPLATE_EDGE.pou ---- *)
FUNCTION_BLOCK L_MC1P_TEMPLATE_EDGE EXTENDS L_MC1P_Template_IntFB
VAR_INPUT
	XEXECUTE : BOOL;
END_VAR
VAR_OUTPUT
	XDONE : BOOL;
	XBUSY : BOOL;
	XCOMMANDABORTED : BOOL;
	XERROR : BOOL;
	EERRORID : L_IE1P_Error;
END_VAR
VAR
	XFIRSTCYCLE : BOOL;
	XEXECUTEOLD : BOOL;
	XRESETOUTPUT : BOOL;
	WFUNID : WORD;
	FUNCTIONTYPE : L_MC1P_TypeFunction;
END_VAR
END_FUNCTION_BLOCK

METHOD ABORT
VAR_IN_OUT
	AXIS : AXIS_REF;
	FBBASE : L_MC1P_Template;
END_VAR
END_METHOD

METHOD CHECKPRECONDITION : BOOL
VAR_OUTPUT
	EERRORID : L_IE1P_Error;
END_VAR
END_METHOD

METHOD CYCLIC
VAR_IN_OUT
	AXIS : AXIS_REF;
	FBBASE : L_MC1P_Template;
END_VAR
END_METHOD

METHOD INIT
VAR_IN_OUT
	AXIS : AXIS_REF;
	FBBASE : L_MC1P_Template;
END_VAR
END_METHOD

METHOD MAIN
VAR_IN_OUT
	AXIS : AXIS_REF;
	FBBASE : L_MC1P_Template;
END_VAR
END_METHOD

METHOD RESETOUTPUTS
END_METHOD

(* ---- L_MC1P_TEMPLATE_FORAXIS.pou ---- *)
FUNCTION_BLOCK L_MC1P_TEMPLATE_FORAXIS
VAR
	XERROROLD : BOOL;
	WERRORIDOLD : WORD;
	XDISABLEERRORRESET : BOOL;
	XDISABLEERRORLOGGING : BOOL;
	DWERRORITFID : DWORD;
	PFBBASEAXIS : POINTER TO AXIS_REF;
	PSINSTANCESTR : POINTER TO STRING;
	DISABLEERRORLOGGING : BOOL;
	DISABLEERRORRESET : BOOL;
END_VAR
END_FUNCTION_BLOCK

METHOD SETINCTANCEINFO
VAR_INPUT
	PSINSTANCENAME : POINTER TO STRING;
	ERRORITFID : DWORD;
END_VAR
END_METHOD

METHOD SETINSTANCEINFOANDAXISPOINTER
VAR_INPUT
	PAXIS : POINTER TO AXIS_REF;
	PSNAME : POINTER TO STRING;
END_VAR
END_METHOD

METHOD UPDATEAXISPOINTER
VAR_INPUT
	PAXIS : POINTER TO AXIS_REF;
END_VAR
END_METHOD

METHOD FB_GETERRORITFID : DWORD
END_METHOD

METHOD FB_GETINSTSTRPOINTER : POINTER TO STRING
END_METHOD

METHOD FB_RESETERROR
VAR_INPUT
	XERROR : BOOL;
	WERRORID : WORD;
END_VAR
END_METHOD

METHOD FB_RESETINT
END_METHOD

METHOD FB_SETERROR
VAR_INPUT
	WERRORID : L_IE1P_Error := 0;
	XSETERRORSTOP : BOOL := FALSE;
END_VAR
END_METHOD

METHOD FB_SETERRORANDREACTION
VAR_INPUT
	WERRORID : L_IE1P_Error := 0;
	EERRORREACTION : L_IE1P_SeverityLevel := L_IE1P_SeverityLevel.NO_RESPONSE;
END_VAR
END_METHOD

METHOD FB_INIT : BOOL
VAR_INPUT
	BINITRETAINS : BOOL;
	BINCOPYCODE : BOOL;
END_VAR
END_METHOD

(* ---- L_MC1P_TEMPLATE_INTERNAL.pou ---- *)
FUNCTION_BLOCK L_MC1P_TEMPLATE_INTERNAL
VAR
	PSINSTANCESTR : POINTER TO STRING;
	DWERRORITFID : DWORD;
	XERROROLD : BOOL;
	WERRORIDOLD : WORD;
END_VAR
END_FUNCTION_BLOCK

METHOD SETINCTANCEINFO
VAR_INPUT
	PSINSTANCENAME : POINTER TO STRING;
	ERRORITFID : DWORD;
END_VAR
END_METHOD

METHOD FB_RESETERROR
VAR_INPUT
	XERROR : BOOL;
	WERRORID : WORD;
END_VAR
VAR_IN_OUT
	AXIS : AXIS_REF;
END_VAR
END_METHOD

METHOD FB_SETERROR
VAR_INPUT
	WERRORID : L_IE1P_Error := 0;
	XSETERRORSTOP : BOOL := FALSE;
END_VAR
VAR_IN_OUT
	AXIS : AXIS_REF;
END_VAR
END_METHOD

METHOD FB_SETLOGWARNING
VAR_INPUT
	WERRORID : L_IE1P_Error := 0;
END_VAR
VAR_IN_OUT
	AXIS : AXIS_REF;
END_VAR
END_METHOD

METHOD FB_INIT : BOOL
VAR_INPUT
	BINITRETAINS : BOOL;
	BINCOPYCODE : BOOL;
END_VAR
END_METHOD

(* ---- L_MC1P_TEMPLATE_INTFB.pou ---- *)
FUNCTION_BLOCK L_MC1P_TEMPLATE_INTFB
END_FUNCTION_BLOCK

METHOD FB_INIT : BOOL
VAR_INPUT
	BINITRETAINS : BOOL;
	BINCOPYCODE : BOOL;
END_VAR
END_METHOD

(* ---- L_MC1P_TEMPLATE_LICENCE_150.pou ---- *)
FUNCTION_BLOCK L_MC1P_TEMPLATE_LICENCE_150 EXTENDS L_MC1P_Template
VAR
	LICHANDLING : L_IMHP_LLMHandling;
END_VAR
END_FUNCTION_BLOCK

METHOD ACTIVATEAPPCREDIT : BOOL
VAR_INPUT
	XACTIVATE : BOOL;
END_VAR
END_METHOD

(* ---- L_MC1P_TEMPLATE_MOVE.pou ---- *)
FUNCTION_BLOCK L_MC1P_TEMPLATE_MOVE EXTENDS L_MC1P_Template_Licence_150
VAR
	GETMOVEBASICP : POINTER TO L_MC1P_MoveBasic;
	PROFILETIME : TIME;
	REMAININGTIMEOFPROFILE : LREAL;
	REMAININGTIMEOFPROFILEAVAILABLE : BOOL;
END_VAR
END_FUNCTION_BLOCK

(* ---- L_MC1P_TIMEAVERAGE.pou ---- *)
FUNCTION_BLOCK L_MC1P_TIMEAVERAGE
VAR_INPUT
	XENABLE : BOOL;
	LRFILTERTIME : LREAL;
	LRCYCLELENGTH : LREAL;
	LRSETPOSIN : LREAL;
	LRSETVELIN : LREAL;
	LRSETACCIN : LREAL;
	LRSETTORQUEIN : LREAL;
	XTRAVERSINGRANGEMODULO : BOOL;
END_VAR
VAR_OUTPUT
	XERROR : BOOL;
	EERRORID : L_IE1P.L_IE1P_Error;
	LRPOSOUT : LREAL;
	LRVELOUT : LREAL;
	LRACCOUT : LREAL;
	LRTORQUEOUT : LREAL;
END_VAR
VAR
	XENABLED : BOOL;
	XENABLEOLD : BOOL;
	XTRAVERSINGRANGEMODULOINT : BOOL;
	XFILTERTIMEINTSETTOONE : BOOL;
	LRTASKCYCLE : LREAL;
	LRHOMINGOFFSETINT : LREAL;
	LRFILTERTIMEINT : LREAL;
	LRINVFILTERTIMEINT : LREAL;
	LRFILTERTIMEPOSTDECIMAL : LREAL;
	LRCYCLELENGTHINT : LREAL;
	LRINVTASKCYCLE : LREAL;
	LRMODCYCLE : LREAL;
	LRFILTEREDPOS : LREAL;
	LRACTPOS : LREAL;
	LROLDPOS : LREAL;
	LRSETPOSINOLD : LREAL;
	LRSETVELINOLD : LREAL;
	LRSETACCINOLD : LREAL;
	LRPOSOUTINT : LREAL;
	WCOUNTER : WORD;
	WFILTERDEPTHINT : WORD;
	IDX : WORD;
	ALRPOSSTATE : ARRAY [0..cwFilterDepthMax] OF LREAL;
	ALRVELSTATE : ARRAY [0..cwFilterDepthMax] OF LREAL;
	ALRACCSTATE : ARRAY [0..cwFilterDepthMax] OF LREAL;
	ALRTORQUESTATE : ARRAY [0..cwFilterDepthMax] OF LREAL;
	ALRPOSROUNDS : ARRAY [0..cwFilterDepthMax] OF LREAL;
	LRSETPOSINTEMP : LREAL;
	LRSETPOSINSAVED : LREAL;
	LRSETVELINSAVED : LREAL;
	LRSETACCINSAVED : LREAL;
	LRSETTORQUEINSAVED : LREAL;
	XFIRSTBUFFERROUND : BOOL;
	WIDX1 : WORD := 0;
	WIDX2 : WORD := 0;
	WSTANDSTILLCNT : WORD := 0;
	CWFILTERDEPTHMAX : WORD := 1023;
END_VAR
END_FUNCTION_BLOCK

METHOD CALCFILTERVALUES
END_METHOD

METHOD DETECTOVERFLOW
VAR_INPUT
	LRACTPOS : LREAL;
	LRPOSOLD : LREAL;
	LRACTCOUNTER : LREAL;
END_VAR
VAR_OUTPUT
	LRNEWCOUNTER : LREAL;
END_VAR
END_METHOD

METHOD ENABLEINIT
END_METHOD

METHOD INITBUFFER
END_METHOD

METHOD READINPUTDATA
END_METHOD

METHOD RESETOUTPUTS
END_METHOD

(* ---- L_MC1P_TORQUECONTROL.pou ---- *)
FUNCTION_BLOCK L_MC1P_TORQUECONTROL EXTENDS L_MC1P_Template_Licence_150
VAR_INPUT
	XEXECUTE : BOOL;
	XCONTINUOUSUPDATE : BOOL := TRUE;
	LRTORQUE : LREAL := 0;
	LRVELOCITYHIGHLIMIT : LREAL := 0;
	LRVELOCITYLOWLIMIT : LREAL := 0;
END_VAR
VAR_OUTPUT
	XBUSY : BOOL;
	XCOMMANDABORTED : BOOL;
	XERROR : BOOL;
	EERRORID : L_IE1P_Error;
END_VAR
VAR
	TF : L_MC1P_TorqueControl_internal;
	VALIDATESPEEDLIMITS : BOOL;
END_VAR
END_FUNCTION_BLOCK

(* ---- L_MC1P_TORQUECONTROL_INTERNAL.pou ---- *)
FUNCTION_BLOCK L_MC1P_TORQUECONTROL_INTERNAL EXTENDS L_MC1P_Template_Edge
VAR_INPUT
	XCONTINUOUSUPDATE : BOOL := TRUE;
	LRTORQUE : LREAL := 0;
	LRVELOCITYLIMITHIGH : LREAL := 0;
	LRVELOCITYLIMITLOW : LREAL := 0;
	XVALIDATESPEEDLIMITS : BOOL := TRUE;
END_VAR
VAR
	XCONTINUOUSUPDATEINT : BOOL;
	LRTORQUE_INT : LREAL := 0;
	LRVELOCITYLIMITHIGH_INT : LREAL := 0;
	LRVELOCITYLIMITLOW_INT : LREAL := 0;
	RG : L_MC1P_RampGeneratorIntern;
	RG_NEG : L_MC1P_RampGeneratorIntern;
	LRSLSDECELERATIONOLD : LREAL;
	EWARNINGID : L_IE1P_Error;
	EWARNINGIDOLD : L_IE1P_Error;
	XSLSWARNINGACTIVE : BOOL;
	XSLSACTIVEOLD : BOOL;
	FUNCTIONTYPE : L_MC1P_TypeFunction;
END_VAR
END_FUNCTION_BLOCK

METHOD ABORT
VAR_IN_OUT
	AXIS : AXIS_REF;
	FBBASE : L_MC1P_Template;
END_VAR
END_METHOD

METHOD CYCLIC
VAR_IN_OUT
	AXIS : AXIS_REF;
	FBBASE : L_MC1P_Template;
END_VAR
END_METHOD

METHOD INIT
VAR_IN_OUT
	AXIS : AXIS_REF;
	FBBASE : L_MC1P_Template;
END_VAR
END_METHOD

METHOD PROCESSTORQUEFOLLOWERSLS
VAR_INPUT
	LRSETUPPERVEL : LREAL;
	LRSETLOWERVEL : LREAL;
END_VAR
VAR_OUTPUT
	LRSETUPPERSLSVELLIMIT : LREAL;
	LRSETLOWERSLSVELLIMIT : LREAL;
END_VAR
VAR_IN_OUT
	AXIS : AXIS_REF;
END_VAR
END_METHOD

(* ---- L_MC1P_TOUCHPROBE_INTERNAL.pou ---- *)
FUNCTION_BLOCK L_MC1P_TOUCHPROBE_INTERNAL EXTENDS L_MC1P_Template_IntFB
VAR_INPUT
	EXECUTE : BOOL;
	WINDOWONLY : BOOL;
	FIRSTPOSITION : LREAL;
	LASTPOSITION : LREAL;
	PAUSEACTIVETP : BOOL;
	XBPB_S131_COMBINATION : BOOL;
END_VAR
VAR_OUTPUT
	DONE : BOOL;
	BUSY : BOOL;
	COMMANDABORTED : BOOL;
	ERROR : BOOL;
	ERRORID : L_IE1P_Error;
	ACTIVATIONLEVEL : BOOL;
	ACTIVATIONLEVELVALID : BOOL;
	VALUESTORED_POSEDGE : BOOL;
	RECPOSITION_POSEDGE : LREAL;
	VALUESTORED_NEGEDGE : BOOL;
	RECPOSITION_NEGEDGE : LREAL;
	NEWVALUESTORED_NEGEDGE : BOOL;
	NEWVALUESTORED_POSEDGE : BOOL;
	TIMESTAMP_POSEDGE : DWORD;
	TIMESTAMP_NEGEDGE : DWORD;
	RECDATA : L_MC1P_TpReceiveData;
END_VAR
VAR
	EXECUTEOLD : BOOL;
	XRESETOUTPUT : BOOL;
	TRIGGERINPUTSAVE : MC_TRIGGER_REF;
	PTPREF : POINTER TO L_MC1P_TPData;
	TPREFSAVE : L_MC1P_TPData;
	XOLDSIGNAL : BOOL;
	WTMP : WORD;
	SNLASTVALIDTPNUMBER : DINT;
	SNTPNUMBER : SINT;
	XWINDOWONLYINT : BOOL;
	LRFIRSTPOSITIONINT : LREAL;
	LRLASTPOSITIONINT : LREAL;
	LRTPPOSITION : LREAL;
	XPOSEDGE : BOOL;
	XNEGEDGE : BOOL;
	WTIMETICKPOSEDGE : WORD;
	WTIMETICKNEGEDGE : WORD;
	DWTPTIMETICKABSCOUNTER : DWORD;
	PFREEENCODERAXIS : POINTER TO _AXIS_REF_ENC;
	LRDELAYCOMPENSATION : LREAL;
	LRTEMP : LREAL;
	LRRECPOSITION_POSEDGE_INT : LREAL;
	LRRECPOSITION_NEGEDGE_INT : LREAL;
	XUSEUNFILTEREDVALUE : BOOL := TRUE;
	DWACTTIMESTAMP : DWORD;
	DWTIMESTAMPABS : DWORD;
	DWTIMESTAMPDIFF : DINT;
	PAXISTPSOURCE : POINTER TO _AXIS_REF_REAL;
END_VAR
END_FUNCTION_BLOCK

METHOD CALCPOSFROMTIMESTAMP : LREAL
VAR_INPUT
	PAXIS : POINTER TO _AXIS_REF_REAL;
	DWTIMESTAMPTP : DWORD;
	XCALCWITHUNFILTEREDVALUES : BOOL := FALSE;
END_VAR
END_METHOD

METHOD CALCTIMESTAMPFROMPOS : DWORD
VAR_INPUT
	PAXIS : POINTER TO _AXIS_REF_REAL;
	DIPOS : DINT;
END_VAR
END_METHOD

METHOD CALCULATEPOSITION : LREAL
VAR_INPUT
	DWDELAY : DWORD;
END_VAR
VAR_IN_OUT
	AXIS : AXIS_REF;
END_VAR
END_METHOD

METHOD CALCULATEPOSITIONTIMETICKS : LREAL
VAR_INPUT
	WTPTIMETICK : WORD;
END_VAR
VAR_IN_OUT
	AXIS : Axis_REF;
END_VAR
END_METHOD

METHOD CHECKINWINDOW : BOOL
VAR_INPUT
	LRPOS : LREAL;
END_VAR
VAR_IN_OUT
	AXIS : Axis_REF;
END_VAR
END_METHOD

METHOD CHECKNEWTP_DIGIN : BOOL
VAR_IN_OUT
	AXIS : AXIS_REF;
END_VAR
END_METHOD

METHOD CHECKNEWTP_DRIVE : BOOL
VAR_IN_OUT
	AXIS : Axis_REF;
END_VAR
END_METHOD

METHOD CHECKNEWTP_ENCODER : BOOL
VAR_INPUT
	PTPAXIS : POINTER TO _AXIS_REF_REAL;
END_VAR
VAR_IN_OUT
	AXIS : Axis_REF;
END_VAR
END_METHOD

METHOD CONVERTFROMUSTONS
VAR_INPUT
	WTIMETICK : WORD;
	WABSTIME : WORD;
END_VAR
VAR_OUTPUT
	DWTIMETICKNS : DWORD;
	DWABSTIMENS : DWORD;
END_VAR
END_METHOD

METHOD MAIN
VAR_IN_OUT
	AXIS : AXIS_REF;
	FBBASE : L_MC1P_Template_ForAxis;
	TRIGGERINPUT : MC_TRIGGER_REF;
END_VAR
END_METHOD

(* ---- L_MC1P_TPAVERAGEDIFF.pou ---- *)
FUNCTION_BLOCK L_MC1P_TPAVERAGEDIFF
VAR_INPUT
	XENABLE : BOOL;
	BYNROFCYCLES : BYTE := 20;
	XTPRECEIVED : BOOL;
	LRSETTPDIFFERENCE : LREAL;
	XTPERRORLIMITED : BOOL;
	LRSETMARKDISTANCE : LREAL;
	LRSETMAXAVERAGE : LREAL := 100;
END_VAR
VAR_OUTPUT
	LRTPERRORAVERAGE : LREAL;
	XAVERAGELIMITED : BOOL;
	LROPTIMISEDGEARFACTOR : LREAL;
END_VAR
VAR
	LRPROCENT : LREAL;
	BYNROFCYCLESINTERNAL : BYTE;
	XTPRECEIVEDOLD : BOOL;
	LRTOTALERROR : LREAL;
	BYCOUNTER : BYTE;
	LROPTIMIZATIONUNCLAMPED : LREAL;
END_VAR
END_FUNCTION_BLOCK

(* ---- L_MC1P_TPCALCDIFF.pou ---- *)
FUNCTION_BLOCK L_MC1P_TPCALCDIFF
VAR_INPUT
	XENABLE : BOOL;
	XTPRECEIVE : BOOL;
	LRACTTPPOSIN : LREAL;
	LRSETTPPOS : LREAL;
	LRCYCLELENGTH : LREAL;
END_VAR
VAR_OUTPUT
	XTPRECEIVED : BOOL;
	LRTPDIFF : LREAL;
	LRTPDIFFTOTAL : LREAL;
END_VAR
VAR
	XINITDONE : BOOL := FALSE;
	XTPRECEIVEOLD : BOOL;
END_VAR
END_FUNCTION_BLOCK

(* ---- L_MC1P_TPCONVERTTP.pou ---- *)
FUNCTION_BLOCK L_MC1P_TPCONVERTTP
VAR_INPUT
	XENABLE : BOOL;
	XTPRECEIVE : BOOL;
	LRACTTPPOSIN : LREAL;
	LRCYCPOSTPAXIS : LREAL;
	LRCYCPOSTARGETAXIS : LREAL;
	LRCYCLELENGTHTPAXIS : LREAL;
	LRCYCLELENGTHTARGETAXIS : LREAL;
END_VAR
VAR_OUTPUT
	XTPRECEIVED : BOOL;
	LRTPACTPOS : LREAL;
	XERROR : BOOL;
	EERRORID : L_IE1P_Error;
END_VAR
VAR
	LRPOSFIFOX : ARRAY [1..20] OF LREAL := [10(0)];
	LRPOSFIFOREG : ARRAY [1..20] OF LREAL := [10(0)];
	BYCOUNTER : INT := 1;
	LRSTACKDIFFERENCE : LREAL;
	LRTPDELTAINMS : LREAL;
	LRDELTAPCT : LREAL;
	XTPRECEIVEDOLD : BOOL;
	LRTEMP : LREAL;
	IDIRECTION : INT;
	LRACTTPPOSINOLD : LREAL;
END_VAR
END_FUNCTION_BLOCK

METHOD SEARCHINSTACKNEGATIVE
END_METHOD

METHOD SEARCHINSTACKPOSITIVE
END_METHOD

(* ---- L_MC1P_TPLIMITDIFF.pou ---- *)
FUNCTION_BLOCK L_MC1P_TPLIMITDIFF
VAR_INPUT
	XTPRECEIVE : BOOL;
	LRSETTPDIFF : LREAL;
	LRSETLIMITMIN : LREAL := -100;
	LRSETLIMITMAX : LREAL := 100;
END_VAR
VAR_OUTPUT
	XTPRECEIVED : BOOL;
	XLIMITACTIVE : BOOL;
	LRTPDIFFLIMITED : LREAL;
END_VAR
VAR
	XTPRECEIVEOLD : BOOL;
	XINITDONE : BOOL;
END_VAR
END_FUNCTION_BLOCK

(* ---- L_MC1P_TPVALUEREADER.pou ---- *)
FUNCTION_BLOCK L_MC1P_TPVALUEREADER
VAR_INPUT
	XCALCULATEPOSITIONVALUEFORSDO : BOOL;
END_VAR
VAR_OUTPUT
	DWVALUE : DWORD;
	XDONE : BOOL;
	XERROR : BOOL;
	XISPDOMAPPED : BOOL;
	XCONFIGURED : BOOL;
END_VAR
VAR
	PAXIS : POINTER TO _AXIS_REF_REAL;
	READSDO : L_DCO.L_DCO_ReadDriveParameter;
	PDWPDOVALUE : POINTER TO DWORD;
	DWDUMMY : DWORD;
END_VAR
END_FUNCTION_BLOCK

METHOD CYCLIC : BOOL
END_METHOD

METHOD EXECUTE : BOOL
END_METHOD

METHOD INIT_FORPDOMAPPING
VAR_INPUT
	PDWVALUE : POINTER TO DWORD;
END_VAR
END_METHOD

METHOD INIT_FORSDOMAPPING
VAR_INPUT
	AXIS : POINTER TO _AXIS_REF_REAL;
	UIINDEX : UINT;
	USISUBINDEX : USINT;
END_VAR
END_METHOD

METHOD INIT_NOTUSED
END_METHOD

METHOD ISEXECUTESET : BOOL
END_METHOD

METHOD RESET
END_METHOD

(* ---- L_MC1P_TPVALUEREADERPDOONLY.pou ---- *)
FUNCTION_BLOCK L_MC1P_TPVALUEREADERPDOONLY
VAR_INPUT
	XCALCULATEPOSITIONVALUEFORSDO : BOOL;
END_VAR
VAR_OUTPUT
	DWVALUE : DWORD;
	XDONE : BOOL;
	XERROR : BOOL;
	XISPDOMAPPED : BOOL;
	XCONFIGURED : BOOL;
END_VAR
VAR
	PAXIS : POINTER TO _AXIS_REF_REAL;
	PDWPDOVALUE : POINTER TO DWORD;
	DWDUMMY : DWORD;
END_VAR
END_FUNCTION_BLOCK

METHOD CYCLIC : BOOL
END_METHOD

METHOD EXECUTE : BOOL
END_METHOD

METHOD INIT_FORPDOMAPPING
VAR_INPUT
	PDWVALUE : POINTER TO DWORD;
END_VAR
END_METHOD

METHOD INIT_NOTUSED
END_METHOD

METHOD ISEXECUTESET : BOOL
END_METHOD

METHOD RESET
END_METHOD

METHOD FB_INIT : BOOL
VAR_INPUT
	BINITRETAINS : BOOL;
	BINCOPYCODE : BOOL;
END_VAR
END_METHOD

(* ---- L_MC1P_TPVALUEWRITER.pou ---- *)
FUNCTION_BLOCK L_MC1P_TPVALUEWRITER
VAR_OUTPUT
	XDONE : BOOL;
	XERROR : BOOL;
	DWVALUE : DWORD;
	XISPDOMAPPED : BOOL;
END_VAR
VAR
	PAXIS : POINTER TO AXIS_REF;
	WRITESDO : L_DCO.L_DCO_WriteDriveParameter;
END_VAR
END_FUNCTION_BLOCK

METHOD CYCLIC : BOOL
END_METHOD

METHOD EXECUTE : BOOL
VAR_INPUT
	DWTHEVALUE : DWORD;
END_VAR
END_METHOD

METHOD INIT_FORPDOMAPPING
END_METHOD

METHOD INIT_FORSDOMAPPING
VAR_INPUT
	AXIS : POINTER TO AXIS_REF;
	UIINDEX : UINT;
	USISUBINDEX : USINT;
	USIDATALENGTH : USINT;
END_VAR
END_METHOD

METHOD RESET
END_METHOD

(* ---- L_MC1P_TPVIRTUALACTPOS.pou ---- *)
FUNCTION_BLOCK L_MC1P_TPVIRTUALACTPOS
VAR_INPUT
	XTPWINDOWOPEN : BOOL;
	XTPRECEIVEDIN : BOOL;
	XMAXTPNOTDETECTED : BOOL;
	LRSETTPPOSIN : LREAL;
	LRACTTPPOSIN : LREAL;
END_VAR
VAR_OUTPUT
	XTPRECEIVEDOUT : BOOL;
	LRACTTPPOS : LREAL;
END_VAR
VAR
	XTPRECEIVEDINOLD : BOOL;
	XFLAGWINDOWOPENANDNOTP : BOOL := FALSE;
	XWINDOWOPENOLD : BOOL;
	XVIRTUALTPACTIVE : BOOL;
END_VAR
END_FUNCTION_BLOCK

(* ---- L_MC1P_TPWINDOW.pou ---- *)
FUNCTION_BLOCK L_MC1P_TPWINDOW
VAR_INPUT
	XENABLE : BOOL;
	LRTPWINDOWSIZE : LREAL;
	LRCYCPOS : LREAL;
	LRCYCVEL : LREAL;
	LRTPSENSORPOS : LREAL;
	XTPRECEIVE : BOOL;
	LRACTTPPOSIN : LREAL;
	LRCYCLELENGTH : LREAL;
	XTEACHMARKWINDOW : BOOL;
	LRSETOFFSETTPWINDOW : LREAL;
	DWMAXTPNOTDETECTED : DWORD;
END_VAR
VAR_OUTPUT
	XTPRECEIVED : BOOL;
	XTPWINDOWOPEN : BOOL;
	XTPWINDOWOPENCOMP : BOOL;
	LRTPDELTAPOSCOMP : LREAL;
	XTPINWINDOW : BOOL;
	XTPNOTINWINDOW : BOOL;
	XTPNOTDETECTED : BOOL;
	XTPSENSORTEACHED : BOOL;
	LRACTTPPOS : LREAL;
	XMAXTPNOTDETECTED : BOOL;
END_VAR
VAR
	XFIRSTSENSOR : BOOL;
	XTPWINDOWOPENOLD : BOOL;
	XTPNOTDETECTEDINTERNAL : BOOL;
	LRLOWERWINDOW : LREAL;
	LRUPPERWINDOW : LREAL;
	LRTPPOSINWINDOWTEST : LREAL;
	XTEACHTPSENSOROLD : BOOL;
	DWMISSEDTPCOUNTER : DWORD;
	LRACTUALREGISTERPOS : LREAL;
	XTPISINWINDOW : BOOL;
	XMISSEDTPDECREMENT : BOOL;
	LRDEADTIMEPOSDIFF : LREAL;
	LRUPPERWINDOWCOMP : LREAL;
	XTPCOMPWINDOWOPEN : BOOL;
	XTPCOMPWINDOWOPENOLD : BOOL := FALSE;
	LRLOWERWINDOWCOMP : LREAL;
	XTPRECEIVEDOLD : BOOL;
	LRACTUALREGISTERPOSOLD : LREAL;
	XTPRECEIVEDINTERNAL : BOOL;
	LRTASKCYCLE : LREAL;
	LRTPWINDOWSIZE_INT : LREAL;
END_VAR
END_FUNCTION_BLOCK

(* ---- L_MC1P_TPWORKER_CIA402.pou ---- *)
FUNCTION_BLOCK L_MC1P_TPWORKER_CIA402
VAR_INPUT
	DWTPSTATUSWORD : DWORD;
	DNTP1POSEDGEVALUE : DINT;
	DNTP1NEGEDGEVALUE : DINT;
	DNTP2POSEDGEVALUE : DINT;
	DNTP2NEGEDGEVALUE : DINT;
	DWTP1POSEDGETIMESTAMP : DWORD;
	DWTP1NEGEDGETIMESTAMP : DWORD;
	DWTP2POSEDGETIMESTAMP : DWORD;
	DWTP2NEGEDGETIMESTAMP : DWORD;
	MAX_TP_INPUTS : SINT := 2;
	XEDGELOGICINDRIVESUPPORTED : BOOL := FALSE;
	XTIMESTAMPSUPPORTED : BOOL := FALSE;
END_VAR
VAR_OUTPUT
	WCTRLWORD : WORD;
END_VAR
VAR
	BINITDONE : BOOL;
	WSTATUSWORD : WORD;
	ANSTATE : ARRAY [1..2] OF BYTE;
	BREADTPSTATUSDONE : BOOL;
	BREADTPSTATUSERROR : BOOL;
	BWRITETPCTRLWORDDONE : BOOL;
	BWRITETPCTRLWORDERROR : BOOL;
	I : SINT;
	PTPREF : POINTER TO L_MC1P_TPData;
	PAXIS : POINTER TO _AXIS_REF_REAL;
	READTPSTATUS : L_MC1P_TpValueReader;
	WRITETPCTRLWORD : L_MC1P_TpValueWriter;
	AREADTPPOSVALUE : ARRAY [1..2] OF L_MC1P_TpValueReader;
	AREADTPNEGVALUE : ARRAY [1..2] OF L_MC1P_TpValueReader;
	AREADTPPOSTIMESTAMP : ARRAY [1..2] OF L_MC1P_TpValueReaderPdoOnly;
	AREADTPNEGTIMESTAMP : ARRAY [1..2] OF L_MC1P_TpValueReaderPdoOnly;
	WCTRLWORDTMP : WORD;
	XSTARTCAPTURINGOLD : ARRAY [1..2] OF BOOL;
	SITPOFFSET : SINT := 0;
	XTIMESTAMPACTIVE : BOOL;
	DWTPSTATUSWORDTMP : DWORD;
	ERRORID_NO_ERROR : INT := 0;
	ERRORID_TP_SELECT : INT := 411;
	ERRORID_TP_MODE : INT := 412;
	ERRORID_TP_ONLY_POS_EDGE : INT := 413;
	ERRORID_TP_EDGE_NOT_AVAILABLE : INT := 414;
	ERRORID_TP_CHANNEL_NOT_FREE : INT := 415;
	ERRORID_TP_MAPPING_FAULT : INT := 416;
	ERRORID_TP_INTERNAL_CHANNEL_NOT_FREE : INT := 417;
	ERRORID_TP_TIMEOUT : INT := 418;
	ERRORID_TP_COMMUNICATION_ERROR : INT := 419;
	ERRORID_TP_ECS_MONITOR_SEL_CHANGED : INT := 420;
	ERRORID_TP_SIGNAL : INT := 421;
	STATE_START : BYTE := 1;
	STATE_WAIT_WRITE_RESPONSE_ENABLE_TP : BYTE := 11;
	STATE_WAIT_WRITE_RESPONSE_DISABLE_TP : BYTE := 21;
	STATE_WAIT_READ_STATUS_RESPONSE : BYTE := 30;
	STATE_WAIT_READ_POS_EDGE_VALUE : BYTE := 40;
	STATE_WAIT_READ_NEG_EDGE_VALUE : BYTE := 45;
	STATE_WAIT_CONTINOUS_MODE_READ_VALUES : BYTE := 50;
	STATE_FINISH_TP_MEASURE : BYTE := 80;
	STATE_ERROR : BYTE := 99;
	STATE_DONE : BYTE := 100;
	TP1 : SINT := 1;
	TP2 : SINT := 2;
END_VAR
END_FUNCTION_BLOCK

METHOD CREATENEWCTRLWORD : WORD
VAR_INPUT
	PTPREF : POINTER TO L_MC1P_TPData;
END_VAR
END_METHOD

METHOD GETPOSITIONSUPPORTED : BOOL
VAR_INPUT
	SNTPINDEX : SINT;
END_VAR
END_METHOD

METHOD GETTIMESTAMP : DWORD
VAR_INPUT
	SNTPINDEX : SINT;
	EDGE : INT;
END_VAR
END_METHOD

METHOD GETTIMESTAMPSUPPORTED : BOOL
VAR_INPUT
	SNTPINDEX : SINT;
END_VAR
END_METHOD

METHOD INIT : BOOL
VAR_INPUT
	PTHEAXIS : POINTER TO _AXIS_REF_REAL;
	WOFFSET : WORD;
	SITPOFFSETINP : SINT := 0;
END_VAR
END_METHOD

METHOD INITVALUE
VAR_INPUT
	LWMAPPINGFLAGPOS : LWORD;
	LWMAPPINGFLAGTIME : LWORD;
	UIINDEXPOS : UINT;
	USISUBINDEXPOS : USINT;
END_VAR
VAR_IN_OUT
	VALREADERPOS : L_MC1P_TpValueReader;
	VALREADERTIME : L_MC1P_TpValueReaderPdoOnly;
	VALPOS : DINT;
	VALTIME : DWORD;
END_VAR
END_METHOD

METHOD TPPROCESSING
VAR_INPUT
	SNTPINDEX : SINT;
END_VAR
END_METHOD

(* ---- L_MC1P_TRACE.pou ---- *)
FUNCTION_BLOCK L_MC1P_TRACE
VAR_INPUT
	DWMASK : DWORD;
	DWTRACEDATA_01 : DWORD;
	DWTRACEDATA_02 : DWORD;
	DWTRACEDATA_03 : DWORD;
	DWTRACEDATA_04 : DWORD;
	DWTRACEDATA_05 : DWORD;
	LRTRACEDATA_06 : LREAL;
	LRTRACEDATA_07 : LREAL;
	LRTRACEDATA_08 : LREAL;
END_VAR
VAR
	WINDEX : DWORD;
	ATRACE : ARRAY [0..L_MC1P_Constants.gc_wTraceMax] OF L_MC1P_TrcElement;
END_VAR
END_FUNCTION_BLOCK

(* ---- L_MC1P_UNIVERSALAXISFACTORY.pou ---- *)
FUNCTION_BLOCK L_MC1P_UNIVERSALAXISFACTORY
VAR
	XMEMINUSE : BOOL;
	EACTIVETYPE : L_MC1P_AxisExtensionTypes;
	PTYPES : POINTER TO L_MC1P_UniversalAxisDataTypes;
	MEMORY : ARRAY [1..cMaxsize] OF BYTE;
	CMAXSIZE : DWORD := (SIZEOF(L_MC1P_UniversalAxisDataTypes) + 16);
END_VAR
END_FUNCTION_BLOCK

METHOD CREATE : L_MC1P_IAxisExtension
VAR_INPUT
	AXISTYPE : L_MC1P_AxisExtensionTypes;
END_VAR
END_METHOD

METHOD DESTROY : BOOL
END_METHOD

METHOD FB_EXIT : BOOL
VAR_INPUT
	BINCOPYCODE : BOOL;
END_VAR
END_METHOD

(* ---- L_MC1P_UNIVERSALENCODERFACTORY.pou ---- *)
FUNCTION_BLOCK L_MC1P_UNIVERSALENCODERFACTORY
VAR
	XMEMINUSE : BOOL;
	EACTIVETYPE : L_MC1P_AxisExtensionTypes;
	PTYPES : POINTER TO L_MC1P_UniversalEncoderDataTypes;
	MEMORY : ARRAY [1..cMaxsize] OF BYTE;
	CMAXSIZE : DWORD := (SIZEOF(L_MC1P_UniversalEncoderDataTypes) + 16);
END_VAR
END_FUNCTION_BLOCK

METHOD CREATE : L_MC1P_IAxisExtension
VAR_INPUT
	AXISTYPE : L_MC1P_AxisExtensionTypes;
END_VAR
END_METHOD

METHOD DESTROY : BOOL
END_METHOD

METHOD FB_EXIT : BOOL
VAR_INPUT
	BINCOPYCODE : BOOL;
END_VAR
END_METHOD

(* ---- L_MC1P_VELOCITYFILTER.pou ---- *)
FUNCTION_BLOCK L_MC1P_VELOCITYFILTER
VAR_INPUT
	XENABLE : BOOL := FALSE;
	LRCYCVEL : LREAL := 0;
	LRFILTERTIME : LREAL := 0;
	LRCOMPVEL : LREAL := 0;
END_VAR
VAR_OUTPUT
	LRSETVELOUT : LREAL := 0;
END_VAR
VAR
	LRINTEGRATOR : LREAL := 0;
	LRSPEEDN0 : LREAL := 0;
	LRSPEEDN1 : LREAL := 0;
	LRCOMPVELINT : LREAL := 0;
	LRTIME : LREAL := 0;
	LRTASKCYCLE : LREAL;
END_VAR
END_FUNCTION_BLOCK

(* ---- L_MC1P_WRITESWLIMIT.pou ---- *)
FUNCTION_BLOCK L_MC1P_WRITESWLIMIT EXTENDS L_MC1P_Template
VAR_INPUT
	XEXECUTE : BOOL;
	XSETSWLIMITPOS : BOOL;
	LRSWLIMITPOS : LREAL;
	XSETSWLIMITNEG : BOOL;
	LRSWLIMITNEG : LREAL;
END_VAR
VAR_OUTPUT
	XDONE : BOOL;
	XERROR : BOOL;
	EERRORID : L_IE1P_Error;
END_VAR
VAR
	LRSWLIMITPOSTMP : LREAL;
	LRSWLIMITNEGTMP : LREAL;
	XEXCECUTEOLD : BOOL := FALSE;
	PLRDUMMY : POINTER TO LREAL;
END_VAR
END_FUNCTION_BLOCK

(* ---- L_MC1P_ZERODETECT.pou ---- *)
FUNCTION_BLOCK L_MC1P_ZERODETECT
VAR_INPUT
	LRSETCYCPOS : LREAL;
	LRCYCLELENGTH : LREAL;
END_VAR
VAR_OUTPUT
	XZERO : BOOL;
	XERROR : BOOL;
	EERRORID : L_IE1P_Error;
END_VAR
VAR
	LRLENGTHINT : LREAL;
	LRPOS : LREAL;
	LRPOSOLD : LREAL;
	LRDIFF : LREAL;
END_VAR
END_FUNCTION_BLOCK

(* ---- MC_ABORTTRIGGER.pou ---- *)
FUNCTION_BLOCK MC_ABORTTRIGGER EXTENDS L_MC1P_Template
VAR_INPUT
	EXECUTE : BOOL;
END_VAR
VAR_OUTPUT
	DONE : BOOL;
	BUSY : BOOL;
	ERROR : BOOL;
	ERRORID : L_IE1P_Error;
END_VAR
VAR_IN_OUT
	TRIGGERINPUT : MC_TRIGGER_REF;
END_VAR
VAR
	ABORTTRIG : L_MC1P_AbortTrigger_Internal;
END_VAR
END_FUNCTION_BLOCK

(* ---- MC_HALT.pou ---- *)
FUNCTION_BLOCK MC_HALT EXTENDS L_MC1P_Template_Move
VAR_INPUT
	EXECUTE : BOOL;
	DECELERATION : LREAL;
	JERK : LREAL;
	BUFFERMODE : MC_BUFFER_MODE;
END_VAR
VAR_OUTPUT
	DONE : BOOL;
	BUSY : BOOL;
	ACTIVE : BOOL;
	COMMANDABORTED : BOOL;
	ERROR : BOOL;
	ERRORID : L_IE1P_Error;
END_VAR
VAR
	HALT : L_MC1P_Halt_Internal;
	XABORTHOMINGALLOWED : BOOL := FALSE;
	ABORTHOMINGALLOWED : BOOL;
	GETMOVEBASICP : POINTER TO L_MC1P_MoveBasic;
END_VAR
END_FUNCTION_BLOCK

(* ---- MC_HALTSUPERIMPOSED.pou ---- *)
FUNCTION_BLOCK MC_HALTSUPERIMPOSED EXTENDS L_MC1P_Template_Move
VAR_INPUT
	EXECUTE : BOOL;
	DECELERATION : LREAL;
	JERK : LREAL;
END_VAR
VAR_OUTPUT
	DONE : BOOL;
	BUSY : BOOL;
	ACTIVE : BOOL;
	COMMANDABORTED : BOOL;
	ERROR : BOOL;
	ERRORID : L_IE1P_Error;
END_VAR
VAR
	FBMB : L_MC1P_MoveBasic := STRUCT(wCalcProfileMode := 1);
	GETMOVEBASICP : POINTER TO L_MC1P_MoveBasic;
END_VAR
END_FUNCTION_BLOCK

(* ---- MC_HOME.pou ---- *)
FUNCTION_BLOCK MC_HOME EXTENDS L_MC1P_Template_Licence_150
VAR_INPUT
	EXECUTE : BOOL;
	POSITION : LREAL;
	BUFFERMODE : MC_BUFFER_MODE;
	HOMEABSSWITCH : BOOL;
	USEEXTPARAMETER : BOOL;
	EXTPARAMETER : L_MC1P_HomeParameter;
	EXTTP : MC_TRIGGER_REF;
	USEPOSITIONINPUT : BOOL := TRUE;
END_VAR
VAR_OUTPUT
	DONE : BOOL;
	BUSY : BOOL;
	ACTIVE : BOOL;
	COMMANDABORTED : BOOL;
	ERROR : BOOL;
	ERRORID : L_IE1P_Error;
END_VAR
VAR
	HOME : L_MC1P_Home_Internal;
END_VAR
END_FUNCTION_BLOCK

(* ---- MC_MOVEABSOLUTE.pou ---- *)
FUNCTION_BLOCK MC_MOVEABSOLUTE EXTENDS L_MC1P_Template_Move
VAR_INPUT
	EXECUTE : BOOL;
	CONTINUOUSUPDATE : BOOL;
	POSITION : LREAL;
	VELOCITY : LREAL;
	ACCELERATION : LREAL;
	DECELERATION : LREAL;
	JERK : LREAL;
	DIRECTION : MC_DIRECTION;
	BUFFERMODE : MC_BUFFER_MODE;
END_VAR
VAR_OUTPUT
	DONE : BOOL;
	BUSY : BOOL;
	ACTIVE : BOOL;
	COMMANDABORTED : BOOL;
	ERROR : BOOL;
	ERRORID : L_IE1P_Error;
END_VAR
VAR
	MOVEABS : L_MC1P_MoveAbsolute_Inernal;
	JERKDEC_INT : LREAL;
	GETMOVEBASICP : POINTER TO L_MC1P_MoveBasic;
	JERKDEC : LREAL;
END_VAR
END_FUNCTION_BLOCK

(* ---- MC_MOVEADDITIVE.pou ---- *)
FUNCTION_BLOCK MC_MOVEADDITIVE EXTENDS L_MC1P_Template_Move
VAR_INPUT
	EXECUTE : BOOL;
	CONTINUOUSUPDATE : BOOL;
	DISTANCE : LREAL;
	VELOCITY : LREAL;
	ACCELERATION : LREAL;
	DECELERATION : LREAL;
	JERK : LREAL;
	BUFFERMODE : MC_BUFFER_MODE;
END_VAR
VAR_OUTPUT
	DONE : BOOL;
	BUSY : BOOL;
	ACTIVE : BOOL;
	COMMANDABORTED : BOOL;
	ERROR : BOOL;
	ERRORID : L_IE1P_Error;
END_VAR
VAR
	FBMB : L_MC1P_MoveBasic := STRUCT(wCalcProfileMode := 1);
	JERKDEC_INT : LREAL;
	GETMOVEBASICP : POINTER TO L_MC1P_MoveBasic;
	JERKDEC : LREAL;
END_VAR
END_FUNCTION_BLOCK

(* ---- MC_MOVECONTINUOUSABSOLUTE.pou ---- *)
FUNCTION_BLOCK MC_MOVECONTINUOUSABSOLUTE EXTENDS L_MC1P_Template_Move
VAR_INPUT
	EXECUTE : BOOL;
	CONTINUOUSUPDATE : BOOL;
	POSITION : LREAL;
	ENDVELOCITY : LREAL;
	VELOCITY : LREAL;
	ACCELERATION : LREAL;
	DECELERATION : LREAL;
	JERK : LREAL;
	DIRECTION : MC_DIRECTION;
	BUFFERMODE : MC_BUFFER_MODE;
END_VAR
VAR_OUTPUT
	INENDVELOCITY : BOOL;
	BUSY : BOOL;
	ACTIVE : BOOL;
	COMMANDABORTED : BOOL;
	ERROR : BOOL;
	ERRORID : L_IE1P_Error;
END_VAR
VAR
	FBMB : L_MC1P_MoveBasic := STRUCT(wCalcProfileMode := 1);
	JERKDEC_INT : LREAL;
	GETMOVEBASICP : POINTER TO L_MC1P_MoveBasic;
	JERKDEC : LREAL;
END_VAR
END_FUNCTION_BLOCK

METHOD RESETEXECUTE
END_METHOD

(* ---- MC_MOVECONTINUOUSRELATIVE.pou ---- *)
FUNCTION_BLOCK MC_MOVECONTINUOUSRELATIVE EXTENDS L_MC1P_Template_Move
VAR_INPUT
	EXECUTE : BOOL;
	CONTINUOUSUPDATE : BOOL;
	DISTANCE : LREAL;
	ENDVELOCITY : LREAL;
	VELOCITY : LREAL;
	ACCELERATION : LREAL;
	DECELERATION : LREAL;
	JERK : LREAL;
	BUFFERMODE : MC_BUFFER_MODE;
END_VAR
VAR_OUTPUT
	INENDVELOCITY : BOOL;
	BUSY : BOOL;
	ACTIVE : BOOL;
	COMMANDABORTED : BOOL;
	ERROR : BOOL;
	ERRORID : L_IE1P_Error;
END_VAR
VAR
	FBMB : L_MC1P_MoveBasic := STRUCT(wCalcProfileMode := 1);
	JERKDEC_INT : LREAL;
	GETMOVEBASICP : POINTER TO L_MC1P_MoveBasic;
	JERKDEC : LREAL;
END_VAR
END_FUNCTION_BLOCK

METHOD RESETEXECUTE
END_METHOD

(* ---- MC_MOVERELATIVE.pou ---- *)
FUNCTION_BLOCK MC_MOVERELATIVE EXTENDS L_MC1P_Template_Move
VAR_INPUT
	EXECUTE : BOOL;
	CONTINUOUSUPDATE : BOOL;
	DISTANCE : LREAL;
	VELOCITY : LREAL;
	ACCELERATION : LREAL;
	DECELERATION : LREAL;
	JERK : LREAL;
	BUFFERMODE : MC_BUFFER_MODE;
END_VAR
VAR_OUTPUT
	DONE : BOOL;
	BUSY : BOOL;
	ACTIVE : BOOL;
	COMMANDABORTED : BOOL;
	ERROR : BOOL;
	ERRORID : L_IE1P_Error;
END_VAR
VAR
	MOVEREL : L_MC1P_MoveRelative_Internal;
	JERKDEC_INT : LREAL;
	GETMOVEBASICP : POINTER TO L_MC1P_MoveBasic;
	JERKDEC : LREAL;
END_VAR
END_FUNCTION_BLOCK

(* ---- MC_MOVESUPERIMPOSED.pou ---- *)
FUNCTION_BLOCK MC_MOVESUPERIMPOSED EXTENDS L_MC1P_Template_Move
VAR_INPUT
	EXECUTE : BOOL;
	CONTINUOUSUPDATE : BOOL;
	DISTANCE : LREAL;
	VELOCITYDIFF : LREAL;
	ACCELERATION : LREAL;
	DECELERATION : LREAL;
	JERK : LREAL;
END_VAR
VAR_OUTPUT
	DONE : BOOL;
	BUSY : BOOL;
	ACTIVE : BOOL;
	COMMANDABORTED : BOOL;
	ERROR : BOOL;
	ERRORID : L_IE1P_Error;
	COVEREDDISTANCE : LREAL;
END_VAR
VAR
	FBMB : L_MC1P_MoveBasic := STRUCT(wCalcProfileMode := 1);
	JERKDEC_INT : LREAL;
	GETMOVEBASICP : POINTER TO L_MC1P_MoveBasic;
	JERKDEC : LREAL;
END_VAR
END_FUNCTION_BLOCK

(* ---- MC_MOVEVELOCITY.pou ---- *)
FUNCTION_BLOCK MC_MOVEVELOCITY EXTENDS L_MC1P_Template_Move
VAR_INPUT
	EXECUTE : BOOL;
	CONTINUOUSUPDATE : BOOL;
	VELOCITY : LREAL;
	ACCELERATION : LREAL;
	DECELERATION : LREAL;
	JERK : LREAL;
	DIRECTION : MC_DIRECTION := MC_DIRECTION.mcPositiveDirection;
	BUFFERMODE : MC_BUFFER_MODE;
END_VAR
VAR_OUTPUT
	INVELOCITY : BOOL;
	BUSY : BOOL;
	ACTIVE : BOOL;
	COMMANDABORTED : BOOL;
	ERROR : BOOL;
	ERRORID : L_IE1P_Error;
END_VAR
VAR
	MOVEVEL : L_MC1P_MoveVelocity_Internal;
	JERKDEC_INT : LREAL;
	GETMOVEBASICP : POINTER TO L_MC1P_MoveBasic;
	JERKDEC : LREAL;
END_VAR
END_FUNCTION_BLOCK

(* ---- MC_POWER.pou ---- *)
FUNCTION_BLOCK MC_POWER EXTENDS L_MC1P_Template
VAR_INPUT
	ENABLE : BOOL;
	ENABLEPOSITIVE : BOOL := TRUE;
	ENABLENEGATIVE : BOOL := TRUE;
END_VAR
VAR_OUTPUT
	STATUS : BOOL;
	VALID : BOOL;
	ERROR : BOOL;
	ERRORID : L_IE1P_Error;
END_VAR
VAR
	WPOWID : WORD := 0;
	ERRORIDOLD : L_IE1P_Error;
END_VAR
END_FUNCTION_BLOCK

(* ---- MC_READACTUALPOSITION.pou ---- *)
FUNCTION_BLOCK MC_READACTUALPOSITION EXTENDS L_MC1P_Template
VAR_INPUT
	ENABLE : BOOL;
END_VAR
VAR_OUTPUT
	VALID : BOOL;
	BUSY : BOOL;
	ERROR : BOOL;
	ERRORID : L_IE1P_Error;
	POSITION : LREAL;
END_VAR
VAR
	XENABLEOLD : BOOL := FALSE;
END_VAR
END_FUNCTION_BLOCK

METHOD FB_RESET : BOOL
END_METHOD

(* ---- MC_READACTUALTORQUE.pou ---- *)
FUNCTION_BLOCK MC_READACTUALTORQUE EXTENDS L_MC1P_Template
VAR_INPUT
	ENABLE : BOOL;
END_VAR
VAR_OUTPUT
	VALID : BOOL;
	BUSY : BOOL;
	ERROR : BOOL;
	ERRORID : L_IE1P_Error;
	TORQUE : LREAL;
END_VAR
VAR
	XENABLEOLD : BOOL := FALSE;
END_VAR
END_FUNCTION_BLOCK

METHOD FB_RESET : BOOL
END_METHOD

(* ---- MC_READACTUALVELOCITY.pou ---- *)
FUNCTION_BLOCK MC_READACTUALVELOCITY EXTENDS L_MC1P_Template
VAR_INPUT
	ENABLE : BOOL;
END_VAR
VAR_OUTPUT
	VALID : BOOL;
	BUSY : BOOL;
	ERROR : BOOL;
	ERRORID : L_IE1P_Error;
	VELOCITY : LREAL;
END_VAR
VAR
	XENABLEOLD : BOOL := FALSE;
END_VAR
END_FUNCTION_BLOCK

METHOD FB_RESET : BOOL
END_METHOD

(* ---- MC_READAXISERROR.pou ---- *)
FUNCTION_BLOCK MC_READAXISERROR EXTENDS L_MC1P_Template
VAR_INPUT
	ENABLE : BOOL;
END_VAR
VAR_OUTPUT
	VALID : BOOL;
	BUSY : BOOL;
	ERROR : BOOL;
	ERRORID : L_IE1P_Error;
	AXISWARNING : BOOL;
	AXISERROR : BOOL;
	AXISERRORID : L_IE1P_Error;
	INSTANCENAME : STRING;
	TIMESTAMP : TIME;
	DRIVEWARNING : BOOL;
	DRIVEERROR : BOOL;
	DRIVEERRORID : DWORD;
END_VAR
VAR
	READ : L_MC1P_ReadAxisError_Internal;
END_VAR
END_FUNCTION_BLOCK

(* ---- MC_READAXISINFO.pou ---- *)
FUNCTION_BLOCK MC_READAXISINFO EXTENDS L_MC1P_Template
VAR_INPUT
	ENABLE : BOOL;
END_VAR
VAR_OUTPUT
	VALID : BOOL;
	BUSY : BOOL;
	ERROR : BOOL;
	ERRORID : L_IE1P_Error;
	HOMEABSSWITCH : BOOL;
	LIMITSWITCHPOS : BOOL;
	LIMITSWITCHNEG : BOOL;
	SIMULATION : BOOL;
	COMMUNICATIONREADY : BOOL;
	READYFORPOWERON : BOOL;
	POWERON : BOOL;
	ISHOMED : BOOL;
	AXISERROR : BOOL;
	AXISWARNING : BOOL;
	DRIVEWARNING : BOOL;
	DRIVEERROR : BOOL;
	SWLIMITSWITCHPOS : BOOL;
	SWLIMITSWITCHNEG : BOOL;
	READYFORMOTION : BOOL;
	STOACTIVE : BOOL;
	VOLTAGEENABLED : BOOL;
	MOTORMAGNETISED : BOOL;
	QSPAPPLACTIVE : BOOL;
	QSPDRIVEACTIVE : BOOL;
END_VAR
VAR
	READ : L_MC1P_ReadAxisInfo_Internal;
END_VAR
END_FUNCTION_BLOCK

(* ---- MC_READBOOLPARAMETER.pou ---- *)
FUNCTION_BLOCK MC_READBOOLPARAMETER EXTENDS L_MC1P_Template
VAR_INPUT
	ENABLE : BOOL;
	PARAMETERNUMBER : DINT;
END_VAR
VAR_OUTPUT
	VALID : BOOL;
	BUSY : BOOL;
	ERROR : BOOL;
	ERRORID : L_IE1P_Error;
	VALUE : BOOL;
END_VAR
VAR
	XENABLEOLD : BOOL := FALSE;
	PARAMETERNUMBEROLD : DINT := 0;
	L_DCO_READDRIVEPARAMETER1 : L_DCO_ReadDriveParameter;
	TIMERREADCYCLE : TON;
	TCYCLETIME : TIME := TIME#1ms;
	XERRORHOLD : BOOL;
	EERRORIDHOLD : L_IE1P_Error;
	READCYCLE : TIME;
END_VAR
END_FUNCTION_BLOCK

METHOD FB_RESET : BOOL
END_METHOD

(* ---- MC_READMOTIONSTATE.pou ---- *)
FUNCTION_BLOCK MC_READMOTIONSTATE EXTENDS L_MC1P_Template
VAR_INPUT
	ENABLE : BOOL;
	SOURCE : MC_SOURCE;
END_VAR
VAR_OUTPUT
	VALID : BOOL;
	BUSY : BOOL;
	ERROR : BOOL;
	ERRORID : L_IE1P_Error;
	CONSTANTVELOCITY : BOOL;
	ACCELERATING : BOOL;
	DECELERATING : BOOL;
	DIRECTIONPOSITIVE : BOOL;
	DIRECTIONNEGATIVE : BOOL;
	INPOSITION : BOOL;
	STANDSTILLSETVELOCITY : BOOL;
	STANDSTILLACTVELOCITY : BOOL;
END_VAR
VAR
	READ : L_MC1P_ReadMotionState_Internal;
END_VAR
END_FUNCTION_BLOCK

(* ---- MC_READPARAMETER.pou ---- *)
FUNCTION_BLOCK MC_READPARAMETER EXTENDS L_MC1P_Template
VAR_INPUT
	ENABLE : BOOL;
	PARAMETERNUMBER : DINT;
END_VAR
VAR_OUTPUT
	VALID : BOOL;
	BUSY : BOOL;
	ERROR : BOOL;
	ERRORID : L_IE1P_Error;
	VALUE : LREAL;
END_VAR
VAR
	READ : L_MC1P_ReadParameter_Internal;
	READCYCLE : TIME;
END_VAR
END_FUNCTION_BLOCK

(* ---- MC_READSTATUS.pou ---- *)
FUNCTION_BLOCK MC_READSTATUS EXTENDS L_MC1P_Template
VAR_INPUT
	ENABLE : BOOL;
END_VAR
VAR_OUTPUT
	VALID : BOOL;
	BUSY : BOOL;
	ERROR : BOOL;
	ERRORID : L_IE1P_Error;
	ERRORSTOP : BOOL;
	DISABLED : BOOL;
	STOPPING : BOOL;
	HOMING : BOOL;
	STANDSTILL : BOOL;
	DISCRETEMOTION : BOOL;
	CONTINUOUSMOTION : BOOL;
	SYNCHRONIZEDMOTION : BOOL;
	CONSTANTVELOCITY : BOOL;
	ACCELERATING : BOOL;
	DECELERATING : BOOL;
	INPOSITION : BOOL;
END_VAR
VAR
	XENABLEOLD : BOOL := FALSE;
END_VAR
END_FUNCTION_BLOCK

METHOD FB_RESET : BOOL
END_METHOD

(* ---- MC_RESET.pou ---- *)
FUNCTION_BLOCK MC_RESET EXTENDS L_MC1P_Template
VAR_INPUT
	EXECUTE : BOOL;
END_VAR
VAR_OUTPUT
	DONE : BOOL;
	BUSY : BOOL;
	ERROR : BOOL;
	ERRORID : L_IE1P_Error;
END_VAR
VAR
	RESET : L_MC1P_Reset_Internal;
END_VAR
END_FUNCTION_BLOCK

(* ---- MC_SETOVERRIDE.pou ---- *)
FUNCTION_BLOCK MC_SETOVERRIDE EXTENDS L_MC1P_Template
VAR_INPUT
	ENABLE : BOOL;
	VELFACTOR : LREAL := 1.0;
	ACCFACTOR : LREAL := 1.0;
	JERKFACTOR : LREAL := 1.0;
END_VAR
VAR_OUTPUT
	ENABLED : BOOL;
	BUSY : BOOL;
	ERROR : BOOL;
	ERRORID : L_IE1P_Error;
END_VAR
VAR
	OVERRIDE : L_MC1P_SetOverride_Internal;
END_VAR
END_FUNCTION_BLOCK

(* ---- MC_SETPOSITION.pou ---- *)
FUNCTION_BLOCK MC_SETPOSITION EXTENDS L_MC1P_Template
VAR_INPUT
	EXECUTE : BOOL;
	POSITION : LREAL;
	RELATIVE : BOOL;
	EXECUTIONMODE : MC_EXECUTION_MODE := MC_EXECUTION_MODE.mcImmediately;
	RESTARTPOSITIONING : BOOL := FALSE;
	USESETTINGSFROMHOMINGMODE : BOOL := FALSE;
END_VAR
VAR_OUTPUT
	DONE : BOOL;
	BUSY : BOOL;
	ERROR : BOOL;
	ERRORID : L_IE1P_Error;
END_VAR
VAR
	XEXECUTEOLD : BOOL;
	XCALLFROMAXESGROUP : BOOL;
	LRDUMMY : LREAL;
	XDISABLELOGMESSAGE : BOOL := FALSE;
	DISABLELOGMESSAGE : BOOL;
END_VAR
END_FUNCTION_BLOCK

METHOD SETCALLFROMAXESGROUP
VAR_INPUT
	XSETCALLFROMAXESGROUP : BOOL;
END_VAR
END_METHOD

(* ---- MC_STOP.pou ---- *)
FUNCTION_BLOCK MC_STOP EXTENDS L_MC1P_Template_Licence_150
VAR_INPUT
	EXECUTE : BOOL;
	DECELERATION : LREAL;
	JERK : LREAL;
END_VAR
VAR_OUTPUT
	DONE : BOOL;
	BUSY : BOOL;
	COMMANDABORTED : BOOL;
	ERROR : BOOL;
	ERRORID : L_IE1P_Error;
END_VAR
VAR
	STOP : L_MC1P_Stop_Internal;
	PROFILETIME : TIME;
	REMAININGTIMEOFPROFILE : LREAL;
	REMAININGTIMEOFPROFILEAVAILABLE : BOOL;
END_VAR
END_FUNCTION_BLOCK

(* ---- MC_TOUCHPROBE.pou ---- *)
FUNCTION_BLOCK MC_TOUCHPROBE EXTENDS L_MC1P_Template
VAR_INPUT
	EXECUTE : BOOL;
	WINDOWONLY : BOOL;
	FIRSTPOSITION : LREAL;
	LASTPOSITION : LREAL;
END_VAR
VAR_OUTPUT
	DONE : BOOL;
	BUSY : BOOL;
	COMMANDABORTED : BOOL;
	ERROR : BOOL;
	ERRORID : L_IE1P_Error;
	ACTIVATIONLEVEL : BOOL;
	ACTIVATIONLEVELVALID : BOOL;
	VALUESTORED_POSEDGE : BOOL;
	RECPOSITION_POSEDGE : LREAL;
	VALUESTORED_NEGEDGE : BOOL;
	RECPOSITION_NEGEDGE : LREAL;
	NEWVALUESTORED_POSEDGE : BOOL;
	NEWVALUESTORED_NEGEDGE : BOOL;
	RECDATA : L_MC1P_TpReceiveData;
END_VAR
VAR_IN_OUT
	TRIGGERINPUT : MC_TRIGGER_REF;
END_VAR
VAR
	TP : L_MC1P_TouchProbe_Internal;
END_VAR
END_FUNCTION_BLOCK

(* ---- MC_WRITEBOOLPARAMETER.pou ---- *)
FUNCTION_BLOCK MC_WRITEBOOLPARAMETER EXTENDS L_MC1P_Template
VAR_INPUT
	EXECUTE : BOOL;
	PARAMETERNUMBER : DINT;
	VALUE : BOOL;
	EXECUTIONMODE : MC_EXECUTION_MODE;
END_VAR
VAR_OUTPUT
	DONE : BOOL;
	BUSY : BOOL;
	ERROR : BOOL;
	ERRORID : L_IE1P_Error;
END_VAR
VAR
	XEXECUTEOLD : BOOL := FALSE;
	XRESETOUTPUT : BOOL := FALSE;
	L_DCO_WRITEDRIVEPARAMETER1 : L_DCO_WriteDriveParameter;
	WERRORID_INT : WORD;
END_VAR
END_FUNCTION_BLOCK

METHOD FB_RESET : BOOL
END_METHOD

(* ---- MC_WRITEPARAMETER.pou ---- *)
FUNCTION_BLOCK MC_WRITEPARAMETER EXTENDS L_MC1P_Template
VAR_INPUT
	EXECUTE : BOOL;
	PARAMETERNUMBER : DINT;
	VALUE : LREAL;
	EXECUTIONMODE : MC_EXECUTION_MODE;
END_VAR
VAR_OUTPUT
	DONE : BOOL;
	BUSY : BOOL;
	ERROR : BOOL;
	ERRORID : L_IE1P_Error;
END_VAR
VAR
	XEXECUTEOLD : BOOL := FALSE;
	XRESETOUTPUT : BOOL := FALSE;
	L_DCO_WRITEDRIVEPARAMETER1 : L_DCO_WriteDriveParameter;
	DWPARAMETERNUMBERINT : DWORD;
	WERRORID_INT : WORD;
END_VAR
END_FUNCTION_BLOCK

METHOD FB_RESET : BOOL
END_METHOD

(* ---- TEXTLIST.pou ---- *)
FUNCTION_BLOCK TEXTLIST
VAR
	M_TEXTLISTFILE : STRING(255);
	_STNAMESPACE : STRING;
END_VAR
END_FUNCTION_BLOCK
